LIN {X 0,Y 187.557,Z 471.713,A -85,B 0,C 180,E1 -25907.007,E2 -25907.007} C_VEL
LIN {X 0,Y 185.924,Z 468.386,A -85,B 0,C 180,E1 -25910.069,E2 -25910.069} C_VEL
LIN {X 0,Y 184.642,Z 465.726,A -85,B 0,C 180,E1 -25913.443,E2 -25913.443} C_VEL
LIN {X 0,Y 183.705,Z 463.049,A -85,B 0,C 180,E1 -25920,E2 -25920} C_VEL
LIN {X 0,Y 183.89,Z 463.764,A -85,B 0,C 180,E1 -25923.286,E2 -25923.286} C_VEL
LIN {X 0,Y 185.707,Z 466.949,A -85,B 0,C 180,E1 -25929.53,E2 -25929.53} C_VEL
LIN {X 0,Y 188.183,Z 471.444,A -85,B 0,C 180,E1 -25934.049,E2 -25934.049} C_VEL
LIN {X 0,Y 190.171,Z 475.16,A -85,B 0,C 180,E1 -25936.781,E2 -25936.781} C_VEL
LIN {X 0,Y 192.965,Z 480.658,A -85,B 0,C 180,E1 -25939.965,E2 -25939.965} C_VEL
LIN {X 0,Y 196.223,Z 487.186,A -85,B 0,C 180,E1 -25943.064,E2 -25943.064} C_VEL
LIN {X 0,Y 198.76,Z 492.903,A -85,B 0,C 180,E1 -25945.217,E2 -25945.217} C_VEL
LIN {X 0,Y 191.942,Z 564.548,A -85,B 0,C 180,E1 -25947.122,E2 -25947.122} C_VEL
LIN {X 0,Y 189.485,Z 579.009,A -85,B 0,C 180,E1 -25947.685,E2 -25947.685} C_VEL
LIN {X 0,Y 185.923,Z 593.535,A -85,B 0,C 180,E1 -25948.495,E2 -25948.495} C_VEL
LIN {X 0,Y 181.708,Z 606.777,A -85,B 0,C 180,E1 -25949.514,E2 -25949.514} C_VEL
LIN {X 0,Y 176.215,Z 620.778,A -85,B 0,C 180,E1 -25950.965,E2 -25950.965} C_VEL
LIN {X 0,Y 170.319,Z 633.449,A -85,B 0,C 180,E1 -25952.729,E2 -25952.729} C_VEL
LIN {X 0,Y 163.721,Z 645.382,A -85,B 0,C 180,E1 -25954.818,E2 -25954.818} C_VEL
LIN {X 0,Y 156.791,Z 656.314,A -85,B 0,C 180,E1 -25957.286,E2 -25957.286} C_VEL
LIN {X 0,Y 149.65,Z 666.389,A -85,B 0,C 180,E1 -25960.258,E2 -25960.258} C_VEL
LIN {X 0,Y 141.683,Z 676.375,A -85,B 0,C 180,E1 -25964.143,E2 -25964.143} C_VEL
LIN {X 0,Y 140.976,Z 677.274,A -85,B 0,C 180,E1 -25964.6,E2 -25964.6} C_VEL
LIN {X 0,Y 138.983,Z 679.517,A -85,B 0,C 180,E1 -25965.653,E2 -25965.653} C_VEL
LIN {X 0,Y 135.25,Z 682.744,A -85,B 0,C 180,E1 -25967.021,E2 -25967.021} C_VEL
LIN {X 0,Y 124.177,Z 690.486,A -85,B 0,C 180,E1 -25970.727,E2 -25970.727} C_VEL
LIN {X 0,Y 120.947,Z 693.059,A -85,B 0,C 180,E1 -25972.711,E2 -25972.711} C_VEL
LIN {X 0,Y 114.755,Z 698.936,A -85,B 0,C 180,E1 -25979.026,E2 -25979.026} C_VEL
LIN {X 0,Y 111.351,Z 702.166,A -85,B 0,C 180,E1 -25983.781,E2 -25983.781} C_VEL
LIN {X 0,Y 107.709,Z 705.681,A -85,B 0,C 180,E1 -25990.959,E2 -25990.959} C_VEL
LIN {X 0,Y 105.674,Z 707.991,A -85,B 0,C 180,E1 -25998.492,E2 -25998.492} C_VEL
LIN {X 0,Y 105.023,Z 709.148,A -85,B 0,C 180,E1 -26006.163,E2 -26006.163} C_VEL
LIN {X 0,Y 105.037,Z 709.297,A -85,B 0,C 180,E1 -26010.001,E2 -26010.001} C_VEL
LIN {X 0,Y 105.023,Z 709.143,A -85,B 0,C 180,E1 -26013.838,E2 -26013.838} C_VEL
LIN {X 0,Y 105.675,Z 707.967,A -85,B 0,C 180,E1 -26021.509,E2 -26021.509} C_VEL
LIN {X 0,Y 107.712,Z 705.634,A -85,B 0,C 180,E1 -26029.041,E2 -26029.041} C_VEL
LIN {X 0,Y 111.352,Z 702.088,A -85,B 0,C 180,E1 -26036.22,E2 -26036.22} C_VEL
LIN {X 0,Y 116.463,Z 697.248,A -85,B 0,C 180,E1 -26042.896,E2 -26042.896} C_VEL
LIN {X 0,Y 123.137,Z 690.987,A -85,B 0,C 180,E1 -26048.89,E2 -26048.89} C_VEL
LIN {X 0,Y 130.236,Z 684.232,A -85,B 0,C 180,E1 -26053.475,E2 -26053.475} C_VEL
LIN {X 0,Y 131.674,Z 683.274,A -85,B 0,C 180,E1 -26054.203,E2 -26054.203} C_VEL
LIN {X 0,Y 137.067,Z 683.812,A -85,B 0,C 180,E1 -26056.959,E2 -26056.959} C_VEL
LIN {X 0,Y 137.658,Z 683.754,A -85,B 0,C 180,E1 -26057.806,E2 -26057.806} C_VEL
LIN {X 0,Y 128.187,Z 680.8,A -85,B 0,C 180,E1 -26062.909,E2 -26062.909} C_VEL
LIN {X 0,Y 117.241,Z 675.145,A -85,B 0,C 180,E1 -26071.832,E2 -26071.832} C_VEL
LIN {X 0,Y 112.757,Z 674.144,A -85,B 0,C 180,E1 -26078.04,E2 -26078.04} C_VEL
LIN {X 0,Y 111.56,Z 673.151,A -85,B 0,C 180,E1 -26081.64,E2 -26081.64} C_VEL
LIN {X 0,Y 109.678,Z 671.783,A -85,B 0,C 180,E1 -26088.917,E2 -26088.917} C_VEL
LIN {X 0,Y 110.012,Z 670.647,A -85,B 0,C 180,E1 -26092.66,E2 -26092.66} C_VEL
LIN {X 0,Y 121.004,Z 665.01,A -85,B 0,C 180,E1 -26116.883,E2 -26116.883} C_VEL
LIN {X 0,Y 127.947,Z 662.916,A -85,B 0,C 180,E1 -26122.613,E2 -26122.613} C_VEL
LIN {X 0,Y 140.954,Z 659.025,A -85,B 0,C 180,E1 -26129.908,E2 -26129.908} C_VEL
LIN {X 0,Y 153.456,Z 654.615,A -85,B 0,C 180,E1 -26134.475,E2 -26134.475} C_VEL
LIN {X 0,Y 153.949,Z 654.617,A -85,B 0,C 180,E1 -26134.741,E2 -26134.741} C_VEL
LIN {X 0,Y 146.413,Z 664.975,A -85,B 0,C 180,E1 -26137.624,E2 -26137.624} C_VEL
LIN {X 0,Y 138.047,Z 675.23,A -85,B 0,C 180,E1 -26141.44,E2 -26141.44} C_VEL
LIN {X 0,Y 130.759,Z 683.495,A -85,B 0,C 180,E1 -26145.675,E2 -26145.675} C_VEL
LIN {X 0,Y 124.795,Z 689.57,A -85,B 0,C 180,E1 -26149.635,E2 -26149.635} C_VEL
LIN {X 0,Y 117.999,Z 696.212,A -85,B 0,C 180,E1 -26155.54,E2 -26155.54} C_VEL
LIN {X 0,Y 112.574,Z 701.409,A -85,B 0,C 180,E1 -26162.08,E2 -26162.08} C_VEL
LIN {X 0,Y 109.405,Z 704.399,A -85,B 0,C 180,E1 -26167.329,E2 -26167.329} C_VEL
LIN {X 0,Y 106.519,Z 707.337,A -85,B 0,C 180,E1 -26174.697,E2 -26174.697} C_VEL
LIN {X 0,Y 105.179,Z 709.095,A -85,B 0,C 180,E1 -26182.32,E2 -26182.32} C_VEL
LIN {X 0,Y 105.034,Z 709.702,A -85,B 0,C 180,E1 -26189.999,E2 -26189.999} C_VEL
LIN {X 0,Y 105.17,Z 709.121,A -85,B 0,C 180,E1 -26197.68,E2 -26197.68} C_VEL
LIN {X 0,Y 106.512,Z 707.397,A -85,B 0,C 180,E1 -26205.303,E2 -26205.303} C_VEL
LIN {X 0,Y 109.375,Z 704.501,A -85,B 0,C 180,E1 -26212.677,E2 -26212.677} C_VEL
LIN {X 0,Y 113.686,Z 700.361,A -85,B 0,C 180,E1 -26219.64,E2 -26219.64} C_VEL
LIN {X 0,Y 119.521,Z 694.867,A -85,B 0,C 180,E1 -26226.016,E2 -26226.016} C_VEL
LIN {X 0,Y 126.588,Z 687.87,A -85,B 0,C 180,E1 -26231.776,E2 -26231.776} C_VEL
LIN {X 0,Y 133.805,Z 680.377,A -85,B 0,C 180,E1 -26236.236,E2 -26236.236} C_VEL
LIN {X 0,Y 140.37,Z 672.723,A -85,B 0,C 180,E1 -26239.776,E2 -26239.776} C_VEL
LIN {X 0,Y 147.577,Z 663.733,A -85,B 0,C 180,E1 -26242.909,E2 -26242.909} C_VEL
LIN {X 0,Y 155.109,Z 653.132,A -85,B 0,C 180,E1 -26245.782,E2 -26245.782} C_VEL
LIN {X 0,Y 162.434,Z 641.573,A -85,B 0,C 180,E1 -26248.115,E2 -26248.115} C_VEL
LIN {X 0,Y 169.184,Z 628.933,A -85,B 0,C 180,E1 -26250.14,E2 -26250.14} C_VEL
LIN {X 0,Y 175.433,Z 615.076,A -85,B 0,C 180,E1 -26251.804,E2 -26251.804} C_VEL
LIN {X 0,Y 180.776,Z 600.557,A -85,B 0,C 180,E1 -26253.092,E2 -26253.092} C_VEL
LIN {X 0,Y 185.145,Z 585.35,A -85,B 0,C 180,E1 -26254.048,E2 -26254.048} C_VEL
LIN {X 0,Y 188.341,Z 569.61,A -85,B 0,C 180,E1 -26254.743,E2 -26254.743} C_VEL
LIN {X 0,Y 190.53,Z 551.213,A -85,B 0,C 180,E1 -26255.288,E2 -26255.288} C_VEL
LIN {X 0,Y 195.388,Z 500.881,A -85,B 0,C 180,E1 -26256.558,E2 -26256.558} C_VEL
LIN {X 0,Y 192.605,Z 493.12,A -85,B 0,C 180,E1 -26259.316,E2 -26259.316} C_VEL
LIN {X 0,Y 189.751,Z 486.108,A -85,B 0,C 180,E1 -26262.556,E2 -26262.556} C_VEL
LIN {X 0,Y 187.846,Z 481.849,A -85,B 0,C 180,E1 -26265.095,E2 -26265.095} C_VEL
LIN {X 0,Y 186.025,Z 477.931,A -85,B 0,C 180,E1 -26268.033,E2 -26268.033} C_VEL
LIN {X 0,Y 184.797,Z 475.213,A -85,B 0,C 180,E1 -26270.56,E2 -26270.56} C_VEL
LIN {X 0,Y 183.646,Z 472.659,A -85,B 0,C 180,E1 -26273.821,E2 -26273.821} C_VEL
LIN {X 0,Y 182.834,Z 470.138,A -85,B 0,C 180,E1 -26280,E2 -26280} C_VEL
LIN {X 0,Y 182.964,Z 470.667,A -85,B 0,C 180,E1 -26282.806,E2 -26282.806} C_VEL
LIN {X 0,Y 184.371,Z 473.499,A -85,B 0,C 180,E1 -26288.494,E2 -26288.494} C_VEL
LIN {X 0,Y 185.251,Z 475.089,A -85,B 0,C 180,E1 -26290.52,E2 -26290.52} C_VEL
LIN {X 0,Y 187.03,Z 478.5,A -85,B 0,C 180,E1 -26293.721,E2 -26293.721} C_VEL
LIN {X 0,Y 189.327,Z 483.029,A -85,B 0,C 180,E1 -26296.946,E2 -26296.946} C_VEL
LIN {X 0,Y 192.711,Z 490.116,A -85,B 0,C 180,E1 -26300.758,E2 -26300.758} C_VEL
LIN {X 0,Y 195.47,Z 496.399,A -85,B 0,C 180,E1 -26303.39,E2 -26303.39} C_VEL
LIN {X 0,Y 189.416,Z 559.8,A -85,B 0,C 180,E1 -26305.06,E2 -26305.06} C_VEL
LIN {X 0,Y 187.005,Z 575.537,A -85,B 0,C 180,E1 -26305.583,E2 -26305.583} C_VEL
LIN {X 0,Y 183.72,Z 589.779,A -85,B 0,C 180,E1 -26306.289,E2 -26306.289} C_VEL
LIN {X 0,Y 179.031,Z 604.867,A -85,B 0,C 180,E1 -26307.357,E2 -26307.357} C_VEL
LIN {X 0,Y 174.055,Z 617.673,A -85,B 0,C 180,E1 -26308.572,E2 -26308.572} C_VEL
LIN {X 0,Y 167.915,Z 630.947,A -85,B 0,C 180,E1 -26310.283,E2 -26310.283} C_VEL
LIN {X 0,Y 161.124,Z 643.241,A -85,B 0,C 180,E1 -26312.317,E2 -26312.317} C_VEL
LIN {X 0,Y 153.87,Z 654.478,A -85,B 0,C 180,E1 -26314.7,E2 -26314.7} C_VEL
LIN {X 0,Y 146.369,Z 664.809,A -85,B 0,C 180,E1 -26317.604,E2 -26317.604} C_VEL
LIN {X 0,Y 139.216,Z 673.563,A -85,B 0,C 180,E1 -26320.779,E2 -26320.779} C_VEL
LIN {X 0,Y 132.788,Z 681.059,A -85,B 0,C 180,E1 -26324.398,E2 -26324.398} C_VEL
LIN {X 0,Y 124.748,Z 689.319,A -85,B 0,C 180,E1 -26329.619,E2 -26329.619} C_VEL
LIN {X 0,Y 120.947,Z 693.059,A -85,B 0,C 180,E1 -26332.711,E2 -26332.711} C_VEL
LIN {X 0,Y 117.868,Z 695.504,A -85,B 0,C 180,E1 -26334.852,E2 -26334.852} C_VEL
LIN {X 0,Y 109.03,Z 700.362,A -85,B 0,C 180,E1 -26339.691,E2 -26339.691} C_VEL
LIN {X 0,Y 104.69,Z 702.688,A -85,B 0,C 180,E1 -26343.013,E2 -26343.013} C_VEL
LIN {X 0,Y 103.243,Z 703.671,A -85,B 0,C 180,E1 -26344.944,E2 -26344.944} C_VEL
LIN {X 0,Y 99.65,Z 706.997,A -85,B 0,C 180,E1 -26353.614,E2 -26353.614} C_VEL
LIN {X 0,Y 98.121,Z 708.726,A -85,B 0,C 180,E1 -26361.764,E2 -26361.764} C_VEL
LIN {X 0,Y 97.93,Z 709.161,A -85,B 0,C 180,E1 -26365.885,E2 -26365.885} C_VEL
LIN {X 0,Y 97.944,Z 709.311,A -85,B 0,C 180,E1 -26370.001,E2 -26370.001} C_VEL
LIN {X 0,Y 97.93,Z 709.156,A -85,B 0,C 180,E1 -26374.116,E2 -26374.116} C_VEL
LIN {X 0,Y 98.697,Z 707.98,A -85,B 0,C 180,E1 -26382.335,E2 -26382.335} C_VEL
LIN {X 0,Y 100.976,Z 705.647,A -85,B 0,C 180,E1 -26390.366,E2 -26390.366} C_VEL
LIN {X 0,Y 104.977,Z 702.102,A -85,B 0,C 180,E1 -26397.946,E2 -26397.946} C_VEL
LIN {X 0,Y 110.518,Z 697.262,A -85,B 0,C 180,E1 -26404.913,E2 -26404.913} C_VEL
LIN {X 0,Y 117.662,Z 691.001,A -85,B 0,C 180,E1 -26411.075,E2 -26411.075} C_VEL
LIN {X 0,Y 125.173,Z 684.243,A -85,B 0,C 180,E1 -26415.715,E2 -26415.715} C_VEL
LIN {X 0,Y 127.95,Z 682.049,A -85,B 0,C 180,E1 -26417.039,E2 -26417.039} C_VEL
LIN {X 0,Y 128.251,Z 682.051,A -85,B 0,C 180,E1 -26417.192,E2 -26417.192} C_VEL
LIN {X 0,Y 127.987,Z 681.841,A -85,B 0,C 180,E1 -26417.919,E2 -26417.919} C_VEL
LIN {X 0,Y 123.687,Z 680.797,A -85,B 0,C 180,E1 -26420.266,E2 -26420.266} C_VEL
LIN {X 0,Y 118.591,Z 680.493,A -85,B 0,C 180,E1 -26423.657,E2 -26423.657} C_VEL
LIN {X 0,Y 112.444,Z 679.282,A -85,B 0,C 180,E1 -26429.999,E2 -26429.999} C_VEL
LIN {X 0,Y 107.401,Z 678.331,A -85,B 0,C 180,E1 -26436.883,E2 -26436.883} C_VEL
LIN {X 0,Y 104.1,Z 676.164,A -85,B 0,C 180,E1 -26448.315,E2 -26448.315} C_VEL
LIN {X 0,Y 104.641,Z 674.305,A -85,B 0,C 180,E1 -26456.149,E2 -26456.149} C_VEL
LIN {X 0,Y 119.117,Z 668.837,A -85,B 0,C 180,E1 -26480.733,E2 -26480.733} C_VEL
LIN {X 0,Y 131.561,Z 665.47,A -85,B 0,C 180,E1 -26488.737,E2 -26488.737} C_VEL
LIN {X 0,Y 141.576,Z 662.528,A -85,B 0,C 180,E1 -26493.097,E2 -26493.097} C_VEL
LIN {X 0,Y 144.111,Z 661.736,A -85,B 0,C 180,E1 -26493.997,E2 -26493.997} C_VEL
LIN {X 0,Y 144.749,Z 661.738,A -85,B 0,C 180,E1 -26494.37,E2 -26494.37} C_VEL
LIN {X 0,Y 135.949,Z 672.398,A -85,B 0,C 180,E1 -26497.967,E2 -26497.967} C_VEL
LIN {X 0,Y 129.046,Z 680.084,A -85,B 0,C 180,E1 -26501.509,E2 -26501.509} C_VEL
LIN {X 0,Y 121.42,Z 687.63,A -85,B 0,C 180,E1 -26506.005,E2 -26506.005} C_VEL
LIN {X 0,Y 113.871,Z 694.667,A -85,B 0,C 180,E1 -26511.888,E2 -26511.888} C_VEL
LIN {X 0,Y 107.647,Z 700.2,A -85,B 0,C 180,E1 -26518.513,E2 -26518.513} C_VEL
LIN {X 0,Y 102.839,Z 704.385,A -85,B 0,C 180,E1 -26525.792,E2 -26525.792} C_VEL
LIN {X 0,Y 99.651,Z 707.323,A -85,B 0,C 180,E1 -26533.614,E2 -26533.614} C_VEL
LIN {X 0,Y 98.12,Z 709.082,A -85,B 0,C 180,E1 -26541.763,E2 -26541.763} C_VEL
LIN {X 0,Y 97.941,Z 709.688,A -85,B 0,C 180,E1 -26549.999,E2 -26549.999} C_VEL
LIN {X 0,Y 98.113,Z 709.107,A -85,B 0,C 180,E1 -26558.236,E2 -26558.236} C_VEL
LIN {X 0,Y 99.643,Z 707.383,A -85,B 0,C 180,E1 -26566.387,E2 -26566.387} C_VEL
LIN {X 0,Y 102.807,Z 704.486,A -85,B 0,C 180,E1 -26574.215,E2 -26574.215} C_VEL
LIN {X 0,Y 107.497,Z 700.345,A -85,B 0,C 180,E1 -26581.535,E2 -26581.535} C_VEL
LIN {X 0,Y 113.815,Z 694.85,A -85,B 0,C 180,E1 -26588.133,E2 -26588.133} C_VEL
LIN {X 0,Y 121.352,Z 687.852,A -85,B 0,C 180,E1 -26594.024,E2 -26594.024} C_VEL
LIN {X 0,Y 128.937,Z 680.358,A -85,B 0,C 180,E1 -26598.544,E2 -26598.544} C_VEL
LIN {X 0,Y 137.073,Z 671.326,A -85,B 0,C 180,E1 -26602.628,E2 -26602.628} C_VEL
LIN {X 0,Y 144.681,Z 662.102,A -85,B 0,C 180,E1 -26605.668,E2 -26605.668} C_VEL
LIN {X 0,Y 153.266,Z 650.21,A -85,B 0,C 180,E1 -26608.654,E2 -26608.654} C_VEL
LIN {X 0,Y 160.848,Z 638.067,A -85,B 0,C 180,E1 -26610.911,E2 -26610.911} C_VEL
LIN {X 0,Y 167.877,Z 624.684,A -85,B 0,C 180,E1 -26612.823,E2 -26612.823} C_VEL
LIN {X 0,Y 173.633,Z 611.575,A -85,B 0,C 180,E1 -26614.236,E2 -26614.236} C_VEL
LIN {X 0,Y 178.792,Z 597.21,A -85,B 0,C 180,E1 -26615.367,E2 -26615.367} C_VEL
LIN {X 0,Y 182.898,Z 582.338,A -85,B 0,C 180,E1 -26616.207,E2 -26616.207} C_VEL
LIN {X 0,Y 185.886,Z 566.815,A -85,B 0,C 180,E1 -26616.817,E2 -26616.817} C_VEL
LIN {X 0,Y 189.95,Z 528.58,A -85,B 0,C 180,E1 -26617.779,E2 -26617.779} C_VEL
LIN {X 0,Y 192.33,Z 504.169,A -85,B 0,C 180,E1 -26618.412,E2 -26618.412} C_VEL
LIN {X 0,Y 189.556,Z 496.227,A -85,B 0,C 180,E1 -26621.527,E2 -26621.527} C_VEL
LIN {X 0,Y 186.843,Z 489.339,A -85,B 0,C 180,E1 -26625.152,E2 -26625.152} C_VEL
LIN {X 0,Y 184.873,Z 484.832,A -85,B 0,C 180,E1 -26628.451,E2 -26628.451} C_VEL
LIN {X 0,Y 183.522,Z 481.695,A -85,B 0,C 180,E1 -26631.466,E2 -26631.466} C_VEL
LIN {X 0,Y 182.585,Z 479.467,A -85,B 0,C 180,E1 -26634.478,E2 -26634.478} C_VEL
LIN {X 0,Y 181.964,Z 477.224,A -85,B 0,C 180,E1 -26640,E2 -26640} C_VEL
LIN {X 0,Y 182.09,Z 477.732,A -85,B 0,C 180,E1 -26642.765,E2 -26642.765} C_VEL
LIN {X 0,Y 183.706,Z 480.982,A -85,B 0,C 180,E1 -26649.036,E2 -26649.036} C_VEL
LIN {X 0,Y 185.598,Z 484.944,A -85,B 0,C 180,E1 -26652.907,E2 -26652.907} C_VEL
LIN {X 0,Y 187.679,Z 489.286,A -85,B 0,C 180,E1 -26656.068,E2 -26656.068} C_VEL
LIN {X 0,Y 190.791,Z 496.28,A -85,B 0,C 180,E1 -26659.851,E2 -26659.851} C_VEL
LIN {X 0,Y 192.425,Z 500.192,A -85,B 0,C 180,E1 -26661.562,E2 -26661.562} C_VEL
LIN {X 0,Y 186.194,Z 562.512,A -85,B 0,C 180,E1 -26663.163,E2 -26663.163} C_VEL
LIN {X 0,Y 183.686,Z 577.382,A -85,B 0,C 180,E1 -26663.671,E2 -26663.671} C_VEL
LIN {X 0,Y 179.963,Z 592.37,A -85,B 0,C 180,E1 -26664.438,E2 -26664.438} C_VEL
LIN {X 0,Y 175.151,Z 606.859,A -85,B 0,C 180,E1 -26665.469,E2 -26665.469} C_VEL
LIN {X 0,Y 169.339,Z 620.846,A -85,B 0,C 180,E1 -26666.836,E2 -26666.836} C_VEL
LIN {X 0,Y 162.674,Z 634.228,A -85,B 0,C 180,E1 -26668.633,E2 -26668.633} C_VEL
LIN {X 0,Y 155.346,Z 646.49,A -85,B 0,C 180,E1 -26670.732,E2 -26670.732} C_VEL
LIN {X 0,Y 147.265,Z 658.124,A -85,B 0,C 180,E1 -26673.368,E2 -26673.368} C_VEL
LIN {X 0,Y 139.601,Z 667.908,A -85,B 0,C 180,E1 -26676.342,E2 -26676.342} C_VEL
LIN {X 0,Y 131.111,Z 677.472,A -85,B 0,C 180,E1 -26680.196,E2 -26680.196} C_VEL
LIN {X 0,Y 124.595,Z 684.398,A -85,B 0,C 180,E1 -26684.013,E2 -26684.013} C_VEL
LIN {X 0,Y 117.454,Z 691.133,A -85,B 0,C 180,E1 -26688.838,E2 -26688.838} C_VEL
LIN {X 0,Y 110.492,Z 697.371,A -85,B 0,C 180,E1 -26695.079,E2 -26695.079} C_VEL
LIN {X 0,Y 104.978,Z 702.182,A -85,B 0,C 180,E1 -26702.055,E2 -26702.055} C_VEL
LIN {X 0,Y 103.243,Z 703.671,A -85,B 0,C 180,E1 -26704.944,E2 -26704.944} C_VEL
LIN {X 0,Y 101.084,Z 705.115,A -85,B 0,C 180,E1 -26707.918,E2 -26707.918} C_VEL
LIN {X 0,Y 96.328,Z 707.026,A -85,B 0,C 180,E1 -26712.844,E2 -26712.844} C_VEL
LIN {X 0,Y 92.819,Z 708.119,A -85,B 0,C 180,E1 -26717.134,E2 -26717.134} C_VEL
LIN {X 0,Y 91.217,Z 708.691,A -85,B 0,C 180,E1 -26720.681,E2 -26720.681} C_VEL
LIN {X 0,Y 91,Z 708.818,A -85,B 0,C 180,E1 -26721.916,E2 -26721.916} C_VEL
LIN {X 0,Y 90.843,Z 709.324,A -85,B 0,C 180,E1 -26730.001,E2 -26730.001} C_VEL
LIN {X 0,Y 90.83,Z 709.17,A -85,B 0,C 180,E1 -26734.438,E2 -26734.438} C_VEL
LIN {X 0,Y 91.753,Z 707.994,A -85,B 0,C 180,E1 -26743.285,E2 -26743.285} C_VEL
LIN {X 0,Y 94.301,Z 705.661,A -85,B 0,C 180,E1 -26751.879,E2 -26751.879} C_VEL
LIN {X 0,Y 98.716,Z 702.115,A -85,B 0,C 180,E1 -26759.892,E2 -26759.892} C_VEL
LIN {X 0,Y 104.732,Z 697.276,A -85,B 0,C 180,E1 -26767.153,E2 -26767.153} C_VEL
LIN {X 0,Y 112.382,Z 691.015,A -85,B 0,C 180,E1 -26773.465,E2 -26773.465} C_VEL
LIN {X 0,Y 119.107,Z 685.31,A -85,B 0,C 180,E1 -26777.507,E2 -26777.507} C_VEL
LIN {X 0,Y 118.001,Z 684.542,A -85,B 0,C 180,E1 -26779.07,E2 -26779.07} C_VEL
LIN {X 0,Y 113.824,Z 684.316,A -85,B 0,C 180,E1 -26781.871,E2 -26781.871} C_VEL
LIN {X 0,Y 104.328,Z 682.804,A -85,B 0,C 180,E1 -26791.865,E2 -26791.865} C_VEL
LIN {X 0,Y 101.937,Z 682.31,A -85,B 0,C 180,E1 -26795.565,E2 -26795.565} C_VEL
LIN {X 0,Y 98.331,Z 680.275,A -85,B 0,C 180,E1 -26807.619,E2 -26807.619} C_VEL
LIN {X 0,Y 99.648,Z 677.815,A -85,B 0,C 180,E1 -26820,E2 -26820} C_VEL
LIN {X 0,Y 113.887,Z 673.365,A -85,B 0,C 180,E1 -26841.732,E2 -26841.732} C_VEL
LIN {X 0,Y 126.706,Z 670.234,A -85,B 0,C 180,E1 -26849.948,E2 -26849.948} C_VEL
LIN {X 0,Y 135.535,Z 668.037,A -85,B 0,C 180,E1 -26853.935,E2 -26853.935} C_VEL
LIN {X 0,Y 126.952,Z 677.401,A -85,B 0,C 180,E1 -26857.677,E2 -26857.677} C_VEL
LIN {X 0,Y 119.812,Z 684.572,A -85,B 0,C 180,E1 -26861.591,E2 -26861.591} C_VEL
LIN {X 0,Y 112.207,Z 691.335,A -85,B 0,C 180,E1 -26866.45,E2 -26866.45} C_VEL
LIN {X 0,Y 104.784,Z 697.596,A -85,B 0,C 180,E1 -26872.868,E2 -26872.868} C_VEL
LIN {X 0,Y 98.776,Z 702.44,A -85,B 0,C 180,E1 -26880.128,E2 -26880.128} C_VEL
LIN {X 0,Y 94.322,Z 705.992,A -85,B 0,C 180,E1 -26888.126,E2 -26888.126} C_VEL
LIN {X 0,Y 91.753,Z 708.333,A -85,B 0,C 180,E1 -26896.715,E2 -26896.715} C_VEL
LIN {X 0,Y 90.8,Z 709.518,A -85,B 0,C 180,E1 -26905.56,E2 -26905.56} C_VEL
LIN {X 0,Y 90.841,Z 709.675,A -85,B 0,C 180,E1 -26909.999,E2 -26909.999} C_VEL
LIN {X 0,Y 91.08,Z 709.093,A -85,B 0,C 180,E1 -26918.877,E2 -26918.877} C_VEL
LIN {X 0,Y 92.822,Z 707.369,A -85,B 0,C 180,E1 -26927.629,E2 -26927.629} C_VEL
LIN {X 0,Y 96.328,Z 704.471,A -85,B 0,C 180,E1 -26935.96,E2 -26935.96} C_VEL
LIN {X 0,Y 101.646,Z 700.148,A -85,B 0,C 180,E1 -26943.931,E2 -26943.931} C_VEL
LIN {X 0,Y 108.26,Z 694.834,A -85,B 0,C 180,E1 -26950.479,E2 -26950.479} C_VEL
LIN {X 0,Y 116.328,Z 687.835,A -85,B 0,C 180,E1 -26956.467,E2 -26956.467} C_VEL
LIN {X 0,Y 123.166,Z 681.497,A -85,B 0,C 180,E1 -26960.383,E2 -26960.383} C_VEL
LIN {X 0,Y 131.582,Z 672.683,A -85,B 0,C 180,E1 -26964.54,E2 -26964.54} C_VEL
LIN {X 0,Y 139.43,Z 663.691,A -85,B 0,C 180,E1 -26967.595,E2 -26967.595} C_VEL
LIN {X 0,Y 147.582,Z 653.085,A -85,B 0,C 180,E1 -26970.351,E2 -26970.351} C_VEL
LIN {X 0,Y 155.38,Z 641.519,A -85,B 0,C 180,E1 -26972.58,E2 -26972.58} C_VEL
LIN {X 0,Y 162.281,Z 629.415,A -85,B 0,C 180,E1 -26974.427,E2 -26974.427} C_VEL
LIN {X 0,Y 168.441,Z 616.732,A -85,B 0,C 180,E1 -26975.882,E2 -26975.882} C_VEL
LIN {X 0,Y 174.056,Z 602.665,A -85,B 0,C 180,E1 -26977.09,E2 -26977.09} C_VEL
LIN {X 0,Y 178.63,Z 588.174,A -85,B 0,C 180,E1 -26977.978,E2 -26977.978} C_VEL
LIN {X 0,Y 182.16,Z 572.756,A -85,B 0,C 180,E1 -26978.653,E2 -26978.653} C_VEL
LIN {X 0,Y 184.496,Z 556.413,A -85,B 0,C 180,E1 -26979.142,E2 -26979.142} C_VEL
LIN {X 0,Y 189.448,Z 507.557,A -85,B 0,C 180,E1 -26980.341,E2 -26980.341} C_VEL
LIN {X 0,Y 187.399,Z 501.513,A -85,B 0,C 180,E1 -26982.912,E2 -26982.912} C_VEL
LIN {X 0,Y 185.313,Z 495.698,A -85,B 0,C 180,E1 -26986.009,E2 -26986.009} C_VEL
LIN {X 0,Y 183.422,Z 491.038,A -85,B 0,C 180,E1 -26989.513,E2 -26989.513} C_VEL
LIN {X 0,Y 182.255,Z 488.018,A -85,B 0,C 180,E1 -26992.522,E2 -26992.522} C_VEL
LIN {X 0,Y 181.521,Z 486.185,A -85,B 0,C 180,E1 -26995.28,E2 -26995.28} C_VEL
LIN {X 0,Y 181.094,Z 484.311,A -85,B 0,C 180,E1 -27000,E2 -27000} C_VEL
LIN {X 0,Y 181.221,Z 484.813,A -85,B 0,C 180,E1 -27002.778,E2 -27002.778} C_VEL
LIN {X 0,Y 182.679,Z 487.972,A -85,B 0,C 180,E1 -27008.713,E2 -27008.713} C_VEL
LIN {X 0,Y 184.456,Z 491.931,A -85,B 0,C 180,E1 -27012.542,E2 -27012.542} C_VEL
LIN {X 0,Y 186.616,Z 496.91,A -85,B 0,C 180,E1 -27015.97,E2 -27015.97} C_VEL
LIN {X 0,Y 189.572,Z 503.969,A -85,B 0,C 180,E1 -27019.667,E2 -27019.667} C_VEL
LIN {X 0,Y 183.191,Z 565.066,A -85,B 0,C 180,E1 -27021.187,E2 -27021.187} C_VEL
LIN {X 0,Y 180.597,Z 579.224,A -85,B 0,C 180,E1 -27021.705,E2 -27021.705} C_VEL
LIN {X 0,Y 176.767,Z 593.692,A -85,B 0,C 180,E1 -27022.425,E2 -27022.425} C_VEL
LIN {X 0,Y 172.217,Z 606.901,A -85,B 0,C 180,E1 -27023.336,E2 -27023.336} C_VEL
LIN {X 0,Y 166.246,Z 620.881,A -85,B 0,C 180,E1 -27024.646,E2 -27024.646} C_VEL
LIN {X 0,Y 159.166,Z 634.654,A -85,B 0,C 180,E1 -27026.448,E2 -27026.448} C_VEL
LIN {X 0,Y 151.84,Z 646.515,A -85,B 0,C 180,E1 -27028.428,E2 -27028.428} C_VEL
LIN {X 0,Y 143.475,Z 658.147,A -85,B 0,C 180,E1 -27030.994,E2 -27030.994} C_VEL
LIN {X 0,Y 135.488,Z 667.929,A -85,B 0,C 180,E1 -27033.907,E2 -27033.907} C_VEL
LIN {X 0,Y 127.097,Z 676.981,A -85,B 0,C 180,E1 -27037.464,E2 -27037.464} C_VEL
LIN {X 0,Y 119.747,Z 684.416,A -85,B 0,C 180,E1 -27041.557,E2 -27041.557} C_VEL
LIN {X 0,Y 112.169,Z 691.15,A -85,B 0,C 180,E1 -27046.433,E2 -27046.433} C_VEL
LIN {X 0,Y 104.705,Z 697.387,A -85,B 0,C 180,E1 -27052.837,E2 -27052.837} C_VEL
LIN {X 0,Y 98.718,Z 702.197,A -85,B 0,C 180,E1 -27060.11,E2 -27060.11} C_VEL
LIN {X 0,Y 94.298,Z 705.711,A -85,B 0,C 180,E1 -27068.121,E2 -27068.121} C_VEL
LIN {X 0,Y 91.753,Z 708.019,A -85,B 0,C 180,E1 -27076.716,E2 -27076.716} C_VEL
LIN {X 0,Y 91,Z 708.818,A -85,B 0,C 180,E1 -27081.916,E2 -27081.916} C_VEL
LIN {X 0,Y 90.041,Z 709.179,A -85,B 0,C 180,E1 -27085.599,E2 -27085.599} C_VEL
LIN {X 0,Y 88.319,Z 709.313,A -85,B 0,C 180,E1 -27089.26,E2 -27089.26} C_VEL
LIN {X 0,Y 84.853,Z 708.996,A -85,B 0,C 180,E1 -27096.908,E2 -27096.908} C_VEL
LIN {X 0,Y 84.278,Z 708.578,A -85,B 0,C 180,E1 -27100.958,E2 -27100.958} C_VEL
LIN {X 0,Y 84.409,Z 708.328,A -85,B 0,C 180,E1 -27102.311,E2 -27102.311} C_VEL
LIN {X 0,Y 86.042,Z 706.988,A -85,B 0,C 180,E1 -27109.071,E2 -27109.071} C_VEL
LIN {X 0,Y 89.952,Z 704.057,A -85,B 0,C 180,E1 -27117.956,E2 -27117.956} C_VEL
LIN {X 0,Y 95.696,Z 699.815,A -85,B 0,C 180,E1 -27126.114,E2 -27126.114} C_VEL
LIN {X 0,Y 103.036,Z 694.347,A -85,B 0,C 180,E1 -27133.008,E2 -27133.008} C_VEL
LIN {X 0,Y 109.3,Z 689.476,A -85,B 0,C 180,E1 -27137.318,E2 -27137.318} C_VEL
LIN {X 0,Y 110.212,Z 687.914,A -85,B 0,C 180,E1 -27139.081,E2 -27139.081} C_VEL
LIN {X 0,Y 104.363,Z 687.333,A -85,B 0,C 180,E1 -27143.912,E2 -27143.912} C_VEL
LIN {X 0,Y 96.419,Z 686.021,A -85,B 0,C 180,E1 -27154.066,E2 -27154.066} C_VEL
LIN {X 0,Y 92.341,Z 683.338,A -85,B 0,C 180,E1 -27171.245,E2 -27171.245} C_VEL
LIN {X 0,Y 96.796,Z 680.537,A -85,B 0,C 180,E1 -27188.35,E2 -27188.35} C_VEL
LIN {X 0,Y 108.523,Z 677.662,A -85,B 0,C 180,E1 -27202.866,E2 -27202.866} C_VEL
LIN {X 0,Y 124.258,Z 674.179,A -85,B 0,C 180,E1 -27212.502,E2 -27212.502} C_VEL
LIN {X 0,Y 125.526,Z 673.895,A -85,B 0,C 180,E1 -27213.086,E2 -27213.086} C_VEL
LIN {X 0,Y 124.864,Z 675.223,A -85,B 0,C 180,E1 -27214.067,E2 -27214.067} C_VEL
LIN {X 0,Y 116.397,Z 683.452,A -85,B 0,C 180,E1 -27218.285,E2 -27218.285} C_VEL
LIN {X 0,Y 109.308,Z 689.527,A -85,B 0,C 180,E1 -27222.319,E2 -27222.319} C_VEL
LIN {X 0,Y 101.037,Z 696.17,A -85,B 0,C 180,E1 -27228.638,E2 -27228.638} C_VEL
LIN {X 0,Y 94.147,Z 701.368,A -85,B 0,C 180,E1 -27235.953,E2 -27235.953} C_VEL
LIN {X 0,Y 89.992,Z 704.358,A -85,B 0,C 180,E1 -27242.057,E2 -27242.057} C_VEL
LIN {X 0,Y 86.047,Z 707.296,A -85,B 0,C 180,E1 -27250.93,E2 -27250.93} C_VEL
LIN {X 0,Y 84.052,Z 709.054,A -85,B 0,C 180,E1 -27260.373,E2 -27260.373} C_VEL
LIN {X 0,Y 83.762,Z 709.661,A -85,B 0,C 180,E1 -27269.999,E2 -27269.999} C_VEL
LIN {X 0,Y 84.047,Z 709.079,A -85,B 0,C 180,E1 -27279.627,E2 -27279.627} C_VEL
LIN {X 0,Y 86.037,Z 707.354,A -85,B 0,C 180,E1 -27289.071,E2 -27289.071} C_VEL
LIN {X 0,Y 89.957,Z 704.456,A -85,B 0,C 180,E1 -27297.953,E2 -27297.953} C_VEL
LIN {X 0,Y 95.559,Z 700.314,A -85,B 0,C 180,E1 -27306.041,E2 -27306.041} C_VEL
LIN {X 0,Y 102.921,Z 694.817,A -85,B 0,C 180,E1 -27313.067,E2 -27313.067} C_VEL
LIN {X 0,Y 111.539,Z 687.817,A -85,B 0,C 180,E1 -27319.122,E2 -27319.122} C_VEL
LIN {X 0,Y 118.71,Z 681.479,A -85,B 0,C 180,E1 -27323.057,E2 -27323.057} C_VEL
LIN {X 0,Y 127.572,Z 672.664,A -85,B 0,C 180,E1 -27327.153,E2 -27327.153} C_VEL
LIN {X 0,Y 135.741,Z 663.669,A -85,B 0,C 180,E1 -27330.138,E2 -27330.138} C_VEL
LIN {X 0,Y 144.198,Z 653.061,A -85,B 0,C 180,E1 -27332.807,E2 -27332.807} C_VEL
LIN {X 0,Y 152.223,Z 641.492,A -85,B 0,C 180,E1 -27334.967,E2 -27334.967} C_VEL
LIN {X 0,Y 159.746,Z 628.619,A -85,B 0,C 180,E1 -27336.831,E2 -27336.831} C_VEL
LIN {X 0,Y 166.419,Z 614.965,A -85,B 0,C 180,E1 -27338.29,E2 -27338.29} C_VEL
LIN {X 0,Y 172.19,Z 600.419,A -85,B 0,C 180,E1 -27339.423,E2 -27339.423} C_VEL
LIN {X 0,Y 176.875,Z 585.168,A -85,B 0,C 180,E1 -27340.255,E2 -27340.255} C_VEL
LIN {X 0,Y 180.179,Z 569.988,A -85,B 0,C 180,E1 -27340.847,E2 -27340.847} C_VEL
LIN {X 0,Y 182.411,Z 553.072,A -85,B 0,C 180,E1 -27341.317,E2 -27341.317} C_VEL
LIN {X 0,Y 186.792,Z 511.201,A -85,B 0,C 180,E1 -27342.291,E2 -27342.291} C_VEL
LIN {X 0,Y 185.055,Z 505.853,A -85,B 0,C 180,E1 -27344.794,E2 -27344.794} C_VEL
LIN {X 0,Y 183.539,Z 501.335,A -85,B 0,C 180,E1 -27347.388,E2 -27347.388} C_VEL
LIN {X 0,Y 182.106,Z 497.425,A -85,B 0,C 180,E1 -27350.419,E2 -27350.419} C_VEL
LIN {X 0,Y 181.116,Z 494.636,A -85,B 0,C 180,E1 -27353.315,E2 -27353.315} C_VEL
LIN {X 0,Y 180.515,Z 492.975,A -85,B 0,C 180,E1 -27355.953,E2 -27355.953} C_VEL
LIN {X 0,Y 180.224,Z 491.396,A -85,B 0,C 180,E1 -27360,E2 -27360} C_VEL
LIN {X 0,Y 180.338,Z 491.855,A -85,B 0,C 180,E1 -27362.652,E2 -27362.652} C_VEL
LIN {X 0,Y 181.595,Z 494.816,A -85,B 0,C 180,E1 -27368.205,E2 -27368.205} C_VEL
LIN {X 0,Y 183.143,Z 498.53,A -85,B 0,C 180,E1 -27371.833,E2 -27371.833} C_VEL
LIN {X 0,Y 185.058,Z 503.289,A -85,B 0,C 180,E1 -27375.135,E2 -27375.135} C_VEL
LIN {X 0,Y 186.902,Z 507.979,A -85,B 0,C 180,E1 -27377.714,E2 -27377.714} C_VEL
LIN {X 0,Y 180.829,Z 564.621,A -85,B 0,C 180,E1 -27379.08,E2 -27379.08} C_VEL
LIN {X 0,Y 178.275,Z 578.411,A -85,B 0,C 180,E1 -27379.536,E2 -27379.536} C_VEL
LIN {X 0,Y 174.183,Z 593.743,A -85,B 0,C 180,E1 -27380.265,E2 -27380.265} C_VEL
LIN {X 0,Y 169.537,Z 606.942,A -85,B 0,C 180,E1 -27381.138,E2 -27381.138} C_VEL
LIN {X 0,Y 163.416,Z 620.915,A -85,B 0,C 180,E1 -27382.386,E2 -27382.386} C_VEL
LIN {X 0,Y 156.281,Z 634.407,A -85,B 0,C 180,E1 -27384.064,E2 -27384.064} C_VEL
LIN {X 0,Y 148.589,Z 646.541,A -85,B 0,C 180,E1 -27386.017,E2 -27386.017} C_VEL
LIN {X 0,Y 139.946,Z 658.169,A -85,B 0,C 180,E1 -27388.498,E2 -27388.498} C_VEL
LIN {X 0,Y 131.635,Z 667.95,A -85,B 0,C 180,E1 -27391.325,E2 -27391.325} C_VEL
LIN {X 0,Y 122.374,Z 677.486,A -85,B 0,C 180,E1 -27395.05,E2 -27395.05} C_VEL
LIN {X 0,Y 115.121,Z 684.434,A -85,B 0,C 180,E1 -27398.889,E2 -27398.889} C_VEL
LIN {X 0,Y 107.093,Z 691.167,A -85,B 0,C 180,E1 -27403.791,E2 -27403.791} C_VEL
LIN {X 0,Y 99.087,Z 697.403,A -85,B 0,C 180,E1 -27410.332,E2 -27410.332} C_VEL
LIN {X 0,Y 92.591,Z 702.212,A -85,B 0,C 180,E1 -27417.906,E2 -27417.906} C_VEL
LIN {X 0,Y 87.704,Z 705.725,A -85,B 0,C 180,E1 -27426.381,E2 -27426.381} C_VEL
LIN {X 0,Y 84.817,Z 708.034,A -85,B 0,C 180,E1 -27435.607,E2 -27435.607} C_VEL
LIN {X 0,Y 83.754,Z 709.189,A -85,B 0,C 180,E1 -27445.187,E2 -27445.187} C_VEL
LIN {X 0,Y 83.764,Z 709.338,A -85,B 0,C 180,E1 -27450.001,E2 -27450.001} C_VEL
LIN {X 0,Y 83.754,Z 709.184,A -85,B 0,C 180,E1 -27454.814,E2 -27454.814} C_VEL
LIN {X 0,Y 84.409,Z 708.328,A -85,B 0,C 180,E1 -27462.311,E2 -27462.311} C_VEL
LIN {X 0,Y 84.574,Z 707.687,A -85,B 0,C 180,E1 -27466.283,E2 -27466.283} C_VEL
LIN {X 0,Y 83.815,Z 706.19,A -85,B 0,C 180,E1 -27472.934,E2 -27472.934} C_VEL
LIN {X 0,Y 83.79,Z 704.692,A -85,B 0,C 180,E1 -27478.283,E2 -27478.283} C_VEL
LIN {X 0,Y 85.292,Z 703.068,A -85,B 0,C 180,E1 -27482.722,E2 -27482.722} C_VEL
LIN {X 0,Y 85.673,Z 702.732,A -85,B 0,C 180,E1 -27483.31,E2 -27483.31} C_VEL
LIN {X 0,Y 91.767,Z 698.659,A -85,B 0,C 180,E1 -27490.616,E2 -27490.616} C_VEL
LIN {X 0,Y 100.176,Z 692.762,A -85,B 0,C 180,E1 -27497.447,E2 -27497.447} C_VEL
LIN {X 0,Y 102.513,Z 691.043,A -85,B 0,C 180,E1 -27498.95,E2 -27498.95} C_VEL
LIN {X 0,Y 90.836,Z 689.485,A -85,B 0,C 180,E1 -27512.341,E2 -27512.341} C_VEL
LIN {X 0,Y 86.18,Z 687.036,A -85,B 0,C 180,E1 -27530.614,E2 -27530.614} C_VEL
LIN {X 0,Y 90.774,Z 684.395,A -85,B 0,C 180,E1 -27548.908,E2 -27548.908} C_VEL
LIN {X 0,Y 103.05,Z 681.714,A -85,B 0,C 180,E1 -27564.155,E2 -27564.155} C_VEL
LIN {X 0,Y 116.736,Z 679.012,A -85,B 0,C 180,E1 -27572.809,E2 -27572.809} C_VEL
LIN {X 0,Y 114.629,Z 681.223,A -85,B 0,C 180,E1 -27574.137,E2 -27574.137} C_VEL
LIN {X 0,Y 107.066,Z 687.588,A -85,B 0,C 180,E1 -27578.028,E2 -27578.028} C_VEL
LIN {X 0,Y 97.878,Z 694.625,A -85,B 0,C 180,E1 -27584.106,E2 -27584.106} C_VEL
LIN {X 0,Y 90.035,Z 700.159,A -85,B 0,C 180,E1 -27591.356,E2 -27591.356} C_VEL
LIN {X 0,Y 83.752,Z 704.345,A -85,B 0,C 180,E1 -27599.768,E2 -27599.768} C_VEL
LIN {X 0,Y 79.313,Z 707.283,A -85,B 0,C 180,E1 -27609.24,E2 -27609.24} C_VEL
LIN {X 0,Y 77.046,Z 709.041,A -85,B 0,C 180,E1 -27619.488,E2 -27619.488} C_VEL
LIN {X 0,Y 76.673,Z 709.647,A -85,B 0,C 180,E1 -27629.999,E2 -27629.999} C_VEL
LIN {X 0,Y 77.042,Z 709.065,A -85,B 0,C 180,E1 -27640.512,E2 -27640.512} C_VEL
LIN {X 0,Y 79.302,Z 707.34,A -85,B 0,C 180,E1 -27650.762,E2 -27650.762} C_VEL
LIN {X 0,Y 83.715,Z 704.441,A -85,B 0,C 180,E1 -27660.245,E2 -27660.245} C_VEL
LIN {X 0,Y 89.882,Z 700.298,A -85,B 0,C 180,E1 -27668.72,E2 -27668.72} C_VEL
LIN {X 0,Y 97.804,Z 694.801,A -85,B 0,C 180,E1 -27675.937,E2 -27675.937} C_VEL
LIN {X 0,Y 107.016,Z 687.8,A -85,B 0,C 180,E1 -27682.005,E2 -27682.005} C_VEL
LIN {X 0,Y 115.797,Z 680.301,A -85,B 0,C 180,E1 -27686.565,E2 -27686.565} C_VEL
LIN {X 0,Y 125.224,Z 671.265,A -85,B 0,C 180,E1 -27690.448,E2 -27690.448} C_VEL
LIN {X 0,Y 133.771,Z 662.037,A -85,B 0,C 180,E1 -27693.269,E2 -27693.269} C_VEL
LIN {X 0,Y 143.31,Z 650.136,A -85,B 0,C 180,E1 -27695.976,E2 -27695.976} C_VEL
LIN {X 0,Y 151.616,Z 637.983,A -85,B 0,C 180,E1 -27697.984,E2 -27697.984} C_VEL
LIN {X 0,Y 159.26,Z 624.585,A -85,B 0,C 180,E1 -27699.675,E2 -27699.675} C_VEL
LIN {X 0,Y 165.478,Z 611.46,A -85,B 0,C 180,E1 -27700.904,E2 -27700.904} C_VEL
LIN {X 0,Y 171.008,Z 597.065,A -85,B 0,C 180,E1 -27701.875,E2 -27701.875} C_VEL
LIN {X 0,Y 175.403,Z 582.145,A -85,B 0,C 180,E1 -27702.574,E2 -27702.574} C_VEL
LIN {X 0,Y 178.632,Z 566.121,A -85,B 0,C 180,E1 -27703.121,E2 -27703.121} C_VEL
LIN {X 0,Y 183.446,Z 523.665,A -85,B 0,C 180,E1 -27704.059,E2 -27704.059} C_VEL
LIN {X 0,Y 184.317,Z 514.847,A -85,B 0,C 180,E1 -27704.339,E2 -27704.339} C_VEL
LIN {X 0,Y 182.369,Z 508.362,A -85,B 0,C 180,E1 -27707.789,E2 -27707.789} C_VEL
LIN {X 0,Y 180.885,Z 503.969,A -85,B 0,C 180,E1 -27711.2,E2 -27711.2} C_VEL
LIN {X 0,Y 180.082,Z 501.463,A -85,B 0,C 180,E1 -27713.839,E2 -27713.839} C_VEL
LIN {X 0,Y 179.574,Z 499.905,A -85,B 0,C 180,E1 -27716.353,E2 -27716.353} C_VEL
LIN {X 0,Y 179.354,Z 498.483,A -85,B 0,C 180,E1 -27720,E2 -27720} C_VEL
LIN {X 0,Y 179.433,Z 498.806,A -85,B 0,C 180,E1 -27722.244,E2 -27722.244} C_VEL
LIN {X 0,Y 180.523,Z 501.67,A -85,B 0,C 180,E1 -27727.691,E2 -27727.691} C_VEL
LIN {X 0,Y 181.87,Z 505.162,A -85,B 0,C 180,E1 -27731.14,E2 -27731.14} C_VEL
LIN {X 0,Y 183.574,Z 509.732,A -85,B 0,C 180,E1 -27734.338,E2 -27734.338} C_VEL
LIN {X 0,Y 184.442,Z 512.24,A -85,B 0,C 180,E1 -27735.728,E2 -27735.728} C_VEL
LIN {X 0,Y 178.531,Z 565.511,A -85,B 0,C 180,E1 -27736.951,E2 -27736.951} C_VEL
LIN {X 0,Y 175.841,Z 579.367,A -85,B 0,C 180,E1 -27737.402,E2 -27737.402} C_VEL
LIN {X 0,Y 171.849,Z 593.795,A -85,B 0,C 180,E1 -27738.041,E2 -27738.041} C_VEL
LIN {X 0,Y 167.107,Z 606.982,A -85,B 0,C 180,E1 -27738.866,E2 -27738.866} C_VEL
LIN {X 0,Y 160.841,Z 620.948,A -85,B 0,C 180,E1 -27740.042,E2 -27740.042} C_VEL
LIN {X 0,Y 153.725,Z 634.084,A -85,B 0,C 180,E1 -27741.589,E2 -27741.589} C_VEL
LIN {X 0,Y 145.602,Z 646.566,A -85,B 0,C 180,E1 -27743.495,E2 -27743.495} C_VEL
LIN {X 0,Y 136.695,Z 658.192,A -85,B 0,C 180,E1 -27745.877,E2 -27745.877} C_VEL
LIN {X 0,Y 128.08,Z 667.97,A -85,B 0,C 180,E1 -27748.605,E2 -27748.605} C_VEL
LIN {X 0,Y 119.751,Z 676.309,A -85,B 0,C 180,E1 -27751.685,E2 -27751.685} C_VEL
LIN {X 0,Y 110.778,Z 684.451,A -85,B 0,C 180,E1 -27756.013,E2 -27756.013} C_VEL
LIN {X 0,Y 102.273,Z 691.183,A -85,B 0,C 180,E1 -27760.897,E2 -27760.897} C_VEL
LIN {X 0,Y 93.694,Z 697.419,A -85,B 0,C 180,E1 -27767.539,E2 -27767.539} C_VEL
LIN {X 0,Y 86.617,Z 702.227,A -85,B 0,C 180,E1 -27775.392,E2 -27775.392} C_VEL
LIN {X 0,Y 81.211,Z 705.74,A -85,B 0,C 180,E1 -27784.362,E2 -27784.362} C_VEL
LIN {X 0,Y 77.928,Z 708.048,A -85,B 0,C 180,E1 -27794.303,E2 -27794.303} C_VEL
LIN {X 0,Y 76.657,Z 709.203,A -85,B 0,C 180,E1 -27804.74,E2 -27804.74} C_VEL
LIN {X 0,Y 76.675,Z 709.352,A -85,B 0,C 180,E1 -27810.001,E2 -27810.001} C_VEL
LIN {X 0,Y 77.046,Z 708.751,A -85,B 0,C 180,E1 -27820.512,E2 -27820.512} C_VEL
LIN {X 0,Y 79.307,Z 707.002,A -85,B 0,C 180,E1 -27830.762,E2 -27830.762} C_VEL
LIN {X 0,Y 83.712,Z 704.071,A -85,B 0,C 180,E1 -27840.248,E2 -27840.248} C_VEL
LIN {X 0,Y 85.673,Z 702.732,A -85,B 0,C 180,E1 -27843.31,E2 -27843.31} C_VEL
LIN {X 0,Y 86.73,Z 701.696,A -85,B 0,C 180,E1 -27845.772,E2 -27845.772} C_VEL
LIN {X 0,Y 87.953,Z 698.06,A -85,B 0,C 180,E1 -27854.276,E2 -27854.276} C_VEL
LIN {X 0,Y 89.641,Z 696.639,A -85,B 0,C 180,E1 -27856.421,E2 -27856.421} C_VEL
LIN {X 0,Y 93.117,Z 694.375,A -85,B 0,C 180,E1 -27859.004,E2 -27859.004} C_VEL
LIN {X 0,Y 91.623,Z 693.445,A -85,B 0,C 180,E1 -27862.147,E2 -27862.147} C_VEL
LIN {X 0,Y 82.969,Z 692.197,A -85,B 0,C 180,E1 -27874.943,E2 -27874.943} C_VEL
LIN {X 0,Y 84.613,Z 687.996,A -85,B 0,C 180,E1 -27909.563,E2 -27909.563} C_VEL
LIN {X 0,Y 101.842,Z 684.785,A -85,B 0,C 180,E1 -27928.886,E2 -27928.886} C_VEL
LIN {X 0,Y 106.578,Z 683.938,A -85,B 0,C 180,E1 -27931.84,E2 -27931.84} C_VEL
LIN {X 0,Y 105.169,Z 685.81,A -85,B 0,C 180,E1 -27933.756,E2 -27933.756} C_VEL
LIN {X 0,Y 95.366,Z 693.012,A -85,B 0,C 180,E1 -27939.303,E2 -27939.303} C_VEL
LIN {X 0,Y 86.535,Z 698.912,A -85,B 0,C 180,E1 -27946.342,E2 -27946.342} C_VEL
LIN {X 0,Y 80.895,Z 702.399,A -85,B 0,C 180,E1 -27952.543,E2 -27952.543} C_VEL
LIN {X 0,Y 74.867,Z 705.951,A -85,B 0,C 180,E1 -27962.006,E2 -27962.006} C_VEL
LIN {X 0,Y 71.097,Z 708.292,A -85,B 0,C 180,E1 -27972.748,E2 -27972.748} C_VEL
LIN {X 0,Y 69.548,Z 709.477,A -85,B 0,C 180,E1 -27984.199,E2 -27984.199} C_VEL
LIN {X 0,Y 69.573,Z 709.634,A -85,B 0,C 180,E1 -27989.999,E2 -27989.999} C_VEL
LIN {X 0,Y 70.046,Z 709.051,A -85,B 0,C 180,E1 -28001.575,E2 -28001.575} C_VEL
LIN {X 0,Y 72.652,Z 707.325,A -85,B 0,C 180,E1 -28012.764,E2 -28012.764} C_VEL
LIN {X 0,Y 77.602,Z 704.426,A -85,B 0,C 180,E1 -28022.914,E2 -28022.914} C_VEL
LIN {X 0,Y 84.432,Z 700.283,A -85,B 0,C 180,E1 -28031.751,E2 -28031.751} C_VEL
LIN {X 0,Y 92.969,Z 694.785,A -85,B 0,C 180,E1 -28039.107,E2 -28039.107} C_VEL
LIN {X 0,Y 102.788,Z 687.783,A -85,B 0,C 180,E1 -28045.132,E2 -28045.132} C_VEL
LIN {X 0,Y 111.981,Z 680.315,A -85,B 0,C 180,E1 -28049.602,E2 -28049.602} C_VEL
LIN {X 0,Y 121.871,Z 671.244,A -85,B 0,C 180,E1 -28053.36,E2 -28053.36} C_VEL
LIN {X 0,Y 130.719,Z 662.015,A -85,B 0,C 180,E1 -28056.062,E2 -28056.062} C_VEL
LIN {X 0,Y 140.567,Z 650.111,A -85,B 0,C 180,E1 -28058.622,E2 -28058.622} C_VEL
LIN {X 0,Y 149.092,Z 637.955,A -85,B 0,C 180,E1 -28060.522,E2 -28060.522} C_VEL
LIN {X 0,Y 156.931,Z 624.551,A -85,B 0,C 180,E1 -28062.112,E2 -28062.112} C_VEL
LIN {X 0,Y 163.293,Z 611.421,A -85,B 0,C 180,E1 -28063.259,E2 -28063.259} C_VEL
LIN {X 0,Y 168.938,Z 597.017,A -85,B 0,C 180,E1 -28064.159,E2 -28064.159} C_VEL
LIN {X 0,Y 173.405,Z 582.079,A -85,B 0,C 180,E1 -28064.819,E2 -28064.819} C_VEL
LIN {X 0,Y 176.64,Z 566.467,A -85,B 0,C 180,E1 -28065.307,E2 -28065.307} C_VEL
LIN {X 0,Y 181.137,Z 527.853,A -85,B 0,C 180,E1 -28066.136,E2 -28066.136} C_VEL
LIN {X 0,Y 182.087,Z 518.948,A -85,B 0,C 180,E1 -28066.362,E2 -28066.362} C_VEL
LIN {X 0,Y 180.857,Z 514.359,A -85,B 0,C 180,E1 -28068.938,E2 -28068.938} C_VEL
LIN {X 0,Y 179.57,Z 510.059,A -85,B 0,C 180,E1 -28072.409,E2 -28072.409} C_VEL
LIN {X 0,Y 178.769,Z 507.233,A -85,B 0,C 180,E1 -28075.914,E2 -28075.914} C_VEL
LIN {X 0,Y 178.486,Z 505.554,A -85,B 0,C 180,E1 -28080,E2 -28080} C_VEL
LIN {X 0,Y 178.563,Z 505.889,A -85,B 0,C 180,E1 -28082.255,E2 -28082.255} C_VEL
LIN {X 0,Y 179.507,Z 508.633,A -85,B 0,C 180,E1 -28087.31,E2 -28087.31} C_VEL
LIN {X 0,Y 180.756,Z 512.11,A -85,B 0,C 180,E1 -28090.732,E2 -28090.732} C_VEL
LIN {X 0,Y 182.202,Z 516.422,A -85,B 0,C 180,E1 -28093.67,E2 -28093.67} C_VEL
LIN {X 0,Y 176.586,Z 565.709,A -85,B 0,C 180,E1 -28094.757,E2 -28094.757} C_VEL
LIN {X 0,Y 173.853,Z 579.441,A -85,B 0,C 180,E1 -28095.172,E2 -28095.172} C_VEL
LIN {X 0,Y 169.788,Z 593.849,A -85,B 0,C 180,E1 -28095.766,E2 -28095.766} C_VEL
LIN {X 0,Y 164.948,Z 607.024,A -85,B 0,C 180,E1 -28096.532,E2 -28096.532} C_VEL
LIN {X 0,Y 158.542,Z 620.983,A -85,B 0,C 180,E1 -28097.624,E2 -28097.624} C_VEL
LIN {X 0,Y 150.848,Z 634.776,A -85,B 0,C 180,E1 -28099.17,E2 -28099.17} C_VEL
LIN {X 0,Y 142.921,Z 646.591,A -85,B 0,C 180,E1 -28100.884,E2 -28100.884} C_VEL
LIN {X 0,Y 133.733,Z 658.214,A -85,B 0,C 180,E1 -28103.123,E2 -28103.123} C_VEL
LIN {X 0,Y 124.829,Z 667.991,A -85,B 0,C 180,E1 -28105.735,E2 -28105.735} C_VEL
LIN {X 0,Y 114.615,Z 677.67,A -85,B 0,C 180,E1 -28109.281,E2 -28109.281} C_VEL
LIN {X 0,Y 105.408,Z 685.497,A -85,B 0,C 180,E1 -28113.548,E2 -28113.548} C_VEL
LIN {X 0,Y 95.337,Z 692.904,A -85,B 0,C 180,E1 -28119.284,E2 -28119.284} C_VEL
LIN {X 0,Y 86.452,Z 698.776,A -85,B 0,C 180,E1 -28126.292,E2 -28126.292} C_VEL
LIN {X 0,Y 80.827,Z 702.243,A -85,B 0,C 180,E1 -28132.508,E2 -28132.508} C_VEL
LIN {X 0,Y 74.842,Z 705.755,A -85,B 0,C 180,E1 -28141.997,E2 -28141.997} C_VEL
LIN {X 0,Y 71.094,Z 708.062,A -85,B 0,C 180,E1 -28152.749,E2 -28152.749} C_VEL
LIN {X 0,Y 69.574,Z 709.217,A -85,B 0,C 180,E1 -28164.203,E2 -28164.203} C_VEL
LIN {X 0,Y 69.576,Z 709.365,A -85,B 0,C 180,E1 -28170.001,E2 -28170.001} C_VEL
LIN {X 0,Y 70.049,Z 708.765,A -85,B 0,C 180,E1 -28181.576,E2 -28181.576} C_VEL
LIN {X 0,Y 72.656,Z 707.015,A -85,B 0,C 180,E1 -28192.764,E2 -28192.764} C_VEL
LIN {X 0,Y 77.602,Z 704.084,A -85,B 0,C 180,E1 -28202.916,E2 -28202.916} C_VEL
LIN {X 0,Y 84.474,Z 699.905,A -85,B 0,C 180,E1 -28211.728,E2 -28211.728} C_VEL
LIN {X 0,Y 89.641,Z 696.639,A -85,B 0,C 180,E1 -28216.421,E2 -28216.421} C_VEL
LIN {X 0,Y 90.16,Z 695.939,A -85,B 0,C 180,E1 -28217.704,E2 -28217.704} C_VEL
LIN {X 0,Y 89.632,Z 695.509,A -85,B 0,C 180,E1 -28219.123,E2 -28219.123} C_VEL
LIN {X 0,Y 87.281,Z 695.263,A -85,B 0,C 180,E1 -28221.617,E2 -28221.617} C_VEL
LIN {X 0,Y 80.136,Z 695.625,A -85,B 0,C 180,E1 -28227.461,E2 -28227.461} C_VEL
LIN {X 0,Y 79.05,Z 695.539,A -85,B 0,C 180,E1 -28229.003,E2 -28229.003} C_VEL
LIN {X 0,Y 73.501,Z 693.618,A -85,B 0,C 180,E1 -28248.976,E2 -28248.976} C_VEL
LIN {X 0,Y 78.333,Z 691.329,A -85,B 0,C 180,E1 -28270.338,E2 -28270.338} C_VEL
LIN {X 0,Y 97.427,Z 688.22,A -85,B 0,C 180,E1 -28291.385,E2 -28291.385} C_VEL
LIN {X 0,Y 95.645,Z 689.858,A -85,B 0,C 180,E1 -28293.134,E2 -28293.134} C_VEL
LIN {X 0,Y 86.096,Z 696.129,A -85,B 0,C 180,E1 -28299.15,E2 -28299.15} C_VEL
LIN {X 0,Y 78.505,Z 700.635,A -85,B 0,C 180,E1 -28305.741,E2 -28305.741} C_VEL
LIN {X 0,Y 71.745,Z 704.317,A -85,B 0,C 180,E1 -28314.001,E2 -28314.001} C_VEL
LIN {X 0,Y 66.124,Z 707.256,A -85,B 0,C 180,E1 -28324.84,E2 -28324.84} C_VEL
LIN {X 0,Y 63.095,Z 709.014,A -85,B 0,C 180,E1 -28337.127,E2 -28337.127} C_VEL
LIN {X 0,Y 62.49,Z 709.62,A -85,B 0,C 180,E1 -28349.999,E2 -28349.999} C_VEL
LIN {X 0,Y 63.091,Z 709.037,A -85,B 0,C 180,E1 -28362.872,E2 -28362.872} C_VEL
LIN {X 0,Y 66.111,Z 707.311,A -85,B 0,C 180,E1 -28375.164,E2 -28375.164} C_VEL
LIN {X 0,Y 71.686,Z 704.411,A -85,B 0,C 180,E1 -28386.031,E2 -28386.031} C_VEL
LIN {X 0,Y 79.232,Z 700.267,A -85,B 0,C 180,E1 -28395.203,E2 -28395.203} C_VEL
LIN {X 0,Y 88.458,Z 694.768,A -85,B 0,C 180,E1 -28402.607,E2 -28402.607} C_VEL
LIN {X 0,Y 96.152,Z 689.67,A -85,B 0,C 180,E1 -28407.199,E2 -28407.199} C_VEL
LIN {X 0,Y 105.752,Z 682.53,A -85,B 0,C 180,E1 -28411.709,E2 -28411.709} C_VEL
LIN {X 0,Y 115.844,Z 673.945,A -85,B 0,C 180,E1 -28415.507,E2 -28415.507} C_VEL
LIN {X 0,Y 126.45,Z 663.605,A -85,B 0,C 180,E1 -28418.582,E2 -28418.582} C_VEL
LIN {X 0,Y 135.76,Z 652.99,A -85,B 0,C 180,E1 -28420.867,E2 -28420.867} C_VEL
LIN {X 0,Y 144.487,Z 641.411,A -85,B 0,C 180,E1 -28422.665,E2 -28422.665} C_VEL
LIN {X 0,Y 152.454,Z 628.795,A -85,B 0,C 180,E1 -28424.2,E2 -28424.2} C_VEL
LIN {X 0,Y 159.76,Z 614.853,A -85,B 0,C 180,E1 -28425.42,E2 -28425.42} C_VEL
LIN {X 0,Y 165.909,Z 600.282,A -85,B 0,C 180,E1 -28426.322,E2 -28426.322} C_VEL
LIN {X 0,Y 170.854,Z 584.987,A -85,B 0,C 180,E1 -28427,E2 -28427} C_VEL
LIN {X 0,Y 174.29,Z 570.059,A -85,B 0,C 180,E1 -28427.468,E2 -28427.468} C_VEL
LIN {X 0,Y 176.731,Z 552.751,A -85,B 0,C 180,E1 -28427.869,E2 -28427.869} C_VEL
LIN {X 0,Y 180.087,Z 523.059,A -85,B 0,C 180,E1 -28428.434,E2 -28428.434} C_VEL
LIN {X 0,Y 179.101,Z 519.229,A -85,B 0,C 180,E1 -28430.969,E2 -28430.969} C_VEL
LIN {X 0,Y 178.172,Z 515.576,A -85,B 0,C 180,E1 -28434.34,E2 -28434.34} C_VEL
LIN {X 0,Y 177.787,Z 514.027,A -85,B 0,C 180,E1 -28436.6,E2 -28436.6} C_VEL
LIN {X 0,Y 177.617,Z 512.628,A -85,B 0,C 180,E1 -28440,E2 -28440} C_VEL
LIN {X 0,Y 177.675,Z 512.883,A -85,B 0,C 180,E1 -28441.983,E2 -28441.983} C_VEL
LIN {X 0,Y 178.463,Z 515.467,A -85,B 0,C 180,E1 -28446.785,E2 -28446.785} C_VEL
LIN {X 0,Y 179.551,Z 518.812,A -85,B 0,C 180,E1 -28450.085,E2 -28450.085} C_VEL
LIN {X 0,Y 180.177,Z 520.85,A -85,B 0,C 180,E1 -28451.572,E2 -28451.572} C_VEL
LIN {X 0,Y 174.881,Z 566.052,A -85,B 0,C 180,E1 -28452.515,E2 -28452.515} C_VEL
LIN {X 0,Y 172.133,Z 579.514,A -85,B 0,C 180,E1 -28452.894,E2 -28452.894} C_VEL
LIN {X 0,Y 168.003,Z 593.902,A -85,B 0,C 180,E1 -28453.442,E2 -28453.442} C_VEL
LIN {X 0,Y 163.069,Z 607.066,A -85,B 0,C 180,E1 -28454.138,E2 -28454.138} C_VEL
LIN {X 0,Y 156.536,Z 621.017,A -85,B 0,C 180,E1 -28455.142,E2 -28455.142} C_VEL
LIN {X 0,Y 148.657,Z 634.806,A -85,B 0,C 180,E1 -28456.571,E2 -28456.571} C_VEL
LIN {X 0,Y 140.546,Z 646.617,A -85,B 0,C 180,E1 -28458.178,E2 -28458.178} C_VEL
LIN {X 0,Y 131.093,Z 658.237,A -85,B 0,C 180,E1 -28460.251,E2 -28460.251} C_VEL
LIN {X 0,Y 121.897,Z 668.011,A -85,B 0,C 180,E1 -28462.709,E2 -28462.709} C_VEL
LIN {X 0,Y 111.445,Z 677.566,A -85,B 0,C 180,E1 -28466.021,E2 -28466.021} C_VEL
LIN {X 0,Y 101.636,Z 685.514,A -85,B 0,C 180,E1 -28470.191,E2 -28470.191} C_VEL
LIN {X 0,Y 90.965,Z 692.921,A -85,B 0,C 180,E1 -28475.785,E2 -28475.785} C_VEL
LIN {X 0,Y 81.425,Z 698.792,A -85,B 0,C 180,E1 -28482.807,E2 -28482.807} C_VEL
LIN {X 0,Y 75.277,Z 702.258,A -85,B 0,C 180,E1 -28489.192,E2 -28489.192} C_VEL
LIN {X 0,Y 68.625,Z 705.769,A -85,B 0,C 180,E1 -28499.2,E2 -28499.2} C_VEL
LIN {X 0,Y 64.295,Z 708.076,A -85,B 0,C 180,E1 -28510.858,E2 -28510.858} C_VEL
LIN {X 0,Y 62.514,Z 709.23,A -85,B 0,C 180,E1 -28523.546,E2 -28523.546} C_VEL
LIN {X 0,Y 62.493,Z 709.379,A -85,B 0,C 180,E1 -28530.001,E2 -28530.001} C_VEL
LIN {X 0,Y 63.094,Z 708.779,A -85,B 0,C 180,E1 -28542.873,E2 -28542.873} C_VEL
LIN {X 0,Y 66.115,Z 707.029,A -85,B 0,C 180,E1 -28555.164,E2 -28555.164} C_VEL
LIN {X 0,Y 71.69,Z 704.098,A -85,B 0,C 180,E1 -28566.03,E2 -28566.03} C_VEL
LIN {X 0,Y 79.276,Z 699.918,A -85,B 0,C 180,E1 -28575.172,E2 -28575.172} C_VEL
LIN {X 0,Y 85.245,Z 696.44,A -85,B 0,C 180,E1 -28580.175,E2 -28580.175} C_VEL
LIN {X 0,Y 84.282,Z 696.11,A -85,B 0,C 180,E1 -28581.875,E2 -28581.875} C_VEL
LIN {X 0,Y 79.05,Z 695.539,A -85,B 0,C 180,E1 -28589.003,E2 -28589.003} C_VEL
LIN {X 0,Y 76.447,Z 695.43,A -85,B 0,C 180,E1 -28592.913,E2 -28592.913} C_VEL
LIN {X 0,Y 67.694,Z 696.312,A -85,B 0,C 180,E1 -28607.086,E2 -28607.086} C_VEL
LIN {X 0,Y 67.108,Z 696.127,A -85,B 0,C 180,E1 -28612.063,E2 -28612.063} C_VEL
LIN {X 0,Y 74.703,Z 693.904,A -85,B 0,C 180,E1 -28636.394,E2 -28636.394} C_VEL
LIN {X 0,Y 87.513,Z 692.169,A -85,B 0,C 180,E1 -28650.336,E2 -28650.336} C_VEL
LIN {X 0,Y 86.175,Z 693.471,A -85,B 0,C 180,E1 -28652.444,E2 -28652.444} C_VEL
LIN {X 0,Y 76.811,Z 698.885,A -85,B 0,C 180,E1 -28658.946,E2 -28658.946} C_VEL
LIN {X 0,Y 70.077,Z 702.372,A -85,B 0,C 180,E1 -28665.409,E2 -28665.409} C_VEL
LIN {X 0,Y 62.61,Z 705.924,A -85,B 0,C 180,E1 -28675.857,E2 -28675.857} C_VEL
LIN {X 0,Y 57.59,Z 708.265,A -85,B 0,C 180,E1 -28688.524,E2 -28688.524} C_VEL
LIN {X 0,Y 55.404,Z 709.45,A -85,B 0,C 180,E1 -28702.711,E2 -28702.711} C_VEL
LIN {X 0,Y 55.39,Z 709.606,A -85,B 0,C 180,E1 -28709.999,E2 -28709.999} C_VEL
LIN {X 0,Y 56.153,Z 709.023,A -85,B 0,C 180,E1 -28724.495,E2 -28724.495} C_VEL
LIN {X 0,Y 59.713,Z 707.296,A -85,B 0,C 180,E1 -28738.084,E2 -28738.084} C_VEL
LIN {X 0,Y 66.018,Z 704.396,A -85,B 0,C 180,E1 -28749.697,E2 -28749.697} C_VEL
LIN {X 0,Y 74.358,Z 700.251,A -85,B 0,C 180,E1 -28759.123,E2 -28759.123} C_VEL
LIN {X 0,Y 84.293,Z 694.752,A -85,B 0,C 180,E1 -28766.486,E2 -28766.486} C_VEL
LIN {X 0,Y 95.339,Z 687.748,A -85,B 0,C 180,E1 -28772.2,E2 -28772.2} C_VEL
LIN {X 0,Y 105.034,Z 680.635,A -85,B 0,C 180,E1 -28776.16,E2 -28776.16} C_VEL
LIN {X 0,Y 116.17,Z 671.204,A -85,B 0,C 180,E1 -28779.67,E2 -28779.67} C_VEL
LIN {X 0,Y 125.61,Z 661.972,A -85,B 0,C 180,E1 -28782.019,E2 -28782.019} C_VEL
LIN {X 0,Y 135.221,Z 651.037,A -85,B 0,C 180,E1 -28784.053,E2 -28784.053} C_VEL
LIN {X 0,Y 144.154,Z 639.068,A -85,B 0,C 180,E1 -28785.689,E2 -28785.689} C_VEL
LIN {X 0,Y 152.337,Z 625.929,A -85,B 0,C 180,E1 -28787.055,E2 -28787.055} C_VEL
LIN {X 0,Y 158.952,Z 613.084,A -85,B 0,C 180,E1 -28788.027,E2 -28788.027} C_VEL
LIN {X 0,Y 164.788,Z 599.135,A -85,B 0,C 180,E1 -28788.789,E2 -28788.789} C_VEL
LIN {X 0,Y 169.61,Z 584.188,A -85,B 0,C 180,E1 -28789.362,E2 -28789.362} C_VEL
LIN {X 0,Y 173.002,Z 569.397,A -85,B 0,C 180,E1 -28789.772,E2 -28789.772} C_VEL
LIN {X 0,Y 175.58,Z 550.754,A -85,B 0,C 180,E1 -28790.188,E2 -28790.188} C_VEL
LIN {X 0,Y 178.277,Z 527.315,A -85,B 0,C 180,E1 -28790.613,E2 -28790.613} C_VEL
LIN {X 0,Y 177.311,Z 522.986,A -85,B 0,C 180,E1 -28794.17,E2 -28794.17} C_VEL
LIN {X 0,Y 176.876,Z 520.993,A -85,B 0,C 180,E1 -28796.898,E2 -28796.898} C_VEL
LIN {X 0,Y 176.743,Z 519.75,A -85,B 0,C 180,E1 -28800,E2 -28800} C_VEL
LIN {X 0,Y 176.791,Z 519.875,A -85,B 0,C 180,E1 -28801.708,E2 -28801.708} C_VEL
LIN {X 0,Y 177.435,Z 522.299,A -85,B 0,C 180,E1 -28806.253,E2 -28806.253} C_VEL
LIN {X 0,Y 178.359,Z 525.496,A -85,B 0,C 180,E1 -28809.403,E2 -28809.403} C_VEL
LIN {X 0,Y 173.492,Z 566.094,A -85,B 0,C 180,E1 -28810.224,E2 -28810.224} C_VEL
LIN {X 0,Y 170.484,Z 580.466,A -85,B 0,C 180,E1 -28810.602,E2 -28810.602} C_VEL
LIN {X 0,Y 166.079,Z 595.219,A -85,B 0,C 180,E1 -28811.12,E2 -28811.12} C_VEL
LIN {X 0,Y 160.65,Z 609.054,A -85,B 0,C 180,E1 -28811.807,E2 -28811.807} C_VEL
LIN {X 0,Y 154.008,Z 622.609,A -85,B 0,C 180,E1 -28812.729,E2 -28812.729} C_VEL
LIN {X 0,Y 146.345,Z 635.52,A -85,B 0,C 180,E1 -28813.978,E2 -28813.978} C_VEL
LIN {X 0,Y 137.674,Z 647.699,A -85,B 0,C 180,E1 -28815.523,E2 -28815.523} C_VEL
LIN {X 0,Y 128.8,Z 658.26,A -85,B 0,C 180,E1 -28817.276,E2 -28817.276} C_VEL
LIN {X 0,Y 119.328,Z 668.032,A -85,B 0,C 180,E1 -28819.552,E2 -28819.552} C_VEL
LIN {X 0,Y 108.499,Z 677.585,A -85,B 0,C 180,E1 -28822.626,E2 -28822.626} C_VEL
LIN {X 0,Y 99.698,Z 684.505,A -85,B 0,C 180,E1 -28826.002,E2 -28826.002} C_VEL
LIN {X 0,Y 89.688,Z 691.234,A -85,B 0,C 180,E1 -28830.463,E2 -28830.463} C_VEL
LIN {X 0,Y 79.189,Z 697.467,A -85,B 0,C 180,E1 -28836.99,E2 -28836.99} C_VEL
LIN {X 0,Y 70.004,Z 702.273,A -85,B 0,C 180,E1 -28845.352,E2 -28845.352} C_VEL
LIN {X 0,Y 62.581,Z 705.784,A -85,B 0,C 180,E1 -28855.84,E2 -28855.84} C_VEL
LIN {X 0,Y 57.586,Z 708.09,A -85,B 0,C 180,E1 -28868.524,E2 -28868.524} C_VEL
LIN {X 0,Y 55.454,Z 709.244,A -85,B 0,C 180,E1 -28882.72,E2 -28882.72} C_VEL
LIN {X 0,Y 55.394,Z 709.393,A -85,B 0,C 180,E1 -28890.001,E2 -28890.001} C_VEL
LIN {X 0,Y 56.155,Z 708.792,A -85,B 0,C 180,E1 -28904.497,E2 -28904.497} C_VEL
LIN {X 0,Y 59.717,Z 707.042,A -85,B 0,C 180,E1 -28918.084,E2 -28918.084} C_VEL
LIN {X 0,Y 66.03,Z 704.112,A -85,B 0,C 180,E1 -28929.69,E2 -28929.69} C_VEL
LIN {X 0,Y 74.401,Z 699.932,A -85,B 0,C 180,E1 -28939.086,E2 -28939.086} C_VEL
LIN {X 0,Y 75.817,Z 699.189,A -85,B 0,C 180,E1 -28940.314,E2 -28940.314} C_VEL
LIN {X 0,Y 76.405,Z 698.508,A -85,B 0,C 180,E1 -28942.103,E2 -28942.103} C_VEL
LIN {X 0,Y 67.681,Z 696.969,A -85,B 0,C 180,E1 -28961.85,E2 -28961.85} C_VEL
LIN {X 0,Y 67.108,Z 696.127,A -85,B 0,C 180,E1 -28972.063,E2 -28972.063} C_VEL
LIN {X 0,Y 67.035,Z 695.944,A -85,B 0,C 180,E1 -28977.107,E2 -28977.107} C_VEL
LIN {X 0,Y 66.294,Z 696.354,A -85,B 0,C 180,E1 -28985.613,E2 -28985.613} C_VEL
LIN {X 0,Y 66.586,Z 696.756,A -85,B 0,C 180,E1 -28992.482,E2 -28992.482} C_VEL
LIN {X 0,Y 68.114,Z 696.768,A -85,B 0,C 180,E1 -28997.361,E2 -28997.361} C_VEL
LIN {X 0,Y 68.956,Z 696.674,A -85,B 0,C 180,E1 -28998.855,E2 -28998.855} C_VEL
LIN {X 0,Y 78.467,Z 695.569,A -85,B 0,C 180,E1 -29009.832,E2 -29009.832} C_VEL
LIN {X 0,Y 76.912,Z 696.584,A -85,B 0,C 180,E1 -29011.519,E2 -29011.519} C_VEL
LIN {X 0,Y 67.674,Z 701.234,A -85,B 0,C 180,E1 -29018.544,E2 -29018.544} C_VEL
LIN {X 0,Y 60.741,Z 704.29,A -85,B 0,C 180,E1 -29026.033,E2 -29026.033} C_VEL
LIN {X 0,Y 53.523,Z 707.228,A -85,B 0,C 180,E1 -29038.315,E2 -29038.315} C_VEL
LIN {X 0,Y 49.286,Z 708.986,A -85,B 0,C 180,E1 -29053.428,E2 -29053.428} C_VEL
LIN {X 0,Y 48.305,Z 709.593,A -85,B 0,C 180,E1 -29069.999,E2 -29069.999} C_VEL
LIN {X 0,Y 49.282,Z 709.009,A -85,B 0,C 180,E1 -29086.571,E2 -29086.571} C_VEL
LIN {X 0,Y 53.507,Z 707.282,A -85,B 0,C 180,E1 -29101.694,E2 -29101.694} C_VEL
LIN {X 0,Y 60.671,Z 704.381,A -85,B 0,C 180,E1 -29114.028,E2 -29114.028} C_VEL
LIN {X 0,Y 69.889,Z 700.236,A -85,B 0,C 180,E1 -29123.558,E2 -29123.558} C_VEL
LIN {X 0,Y 80.558,Z 694.735,A -85,B 0,C 180,E1 -29130.74,E2 -29130.74} C_VEL
LIN {X 0,Y 92.221,Z 687.73,A -85,B 0,C 180,E1 -29136.134,E2 -29136.134} C_VEL
LIN {X 0,Y 103.005,Z 680.094,A -85,B 0,C 180,E1 -29140.053,E2 -29140.053} C_VEL
LIN {X 0,Y 113.889,Z 671.184,A -85,B 0,C 180,E1 -29143.035,E2 -29143.035} C_VEL
LIN {X 0,Y 123.592,Z 661.95,A -85,B 0,C 180,E1 -29145.17,E2 -29145.17} C_VEL
LIN {X 0,Y 133.444,Z 651.013,A -85,B 0,C 180,E1 -29146.988,E2 -29146.988} C_VEL
LIN {X 0,Y 142.768,Z 638.745,A -85,B 0,C 180,E1 -29148.505,E2 -29148.505} C_VEL
LIN {X 0,Y 150.903,Z 625.897,A -85,B 0,C 180,E1 -29149.688,E2 -29149.688} C_VEL
LIN {X 0,Y 157.633,Z 613.046,A -85,B 0,C 180,E1 -29150.551,E2 -29150.551} C_VEL
LIN {X 0,Y 163.556,Z 599.088,A -85,B 0,C 180,E1 -29151.228,E2 -29151.228} C_VEL
LIN {X 0,Y 168.445,Z 584.126,A -85,B 0,C 180,E1 -29151.733,E2 -29151.733} C_VEL
LIN {X 0,Y 171.936,Z 569.028,A -85,B 0,C 180,E1 -29152.112,E2 -29152.112} C_VEL
LIN {X 0,Y 174.503,Z 550.691,A -85,B 0,C 180,E1 -29152.48,E2 -29152.48} C_VEL
LIN {X 0,Y 176.691,Z 532.02,A -85,B 0,C 180,E1 -29152.791,E2 -29152.791} C_VEL
LIN {X 0,Y 176.131,Z 528.993,A -85,B 0,C 180,E1 -29155.737,E2 -29155.737} C_VEL
LIN {X 0,Y 175.89,Z 527.578,A -85,B 0,C 180,E1 -29158.139,E2 -29158.139} C_VEL
LIN {X 0,Y 175.872,Z 526.84,A -85,B 0,C 180,E1 -29160,E2 -29160} C_VEL
LIN {X 0,Y 175.92,Z 526.977,A -85,B 0,C 180,E1 -29161.717,E2 -29161.717} C_VEL
LIN {X 0,Y 176.45,Z 529.259,A -85,B 0,C 180,E1 -29165.858,E2 -29165.858} C_VEL
LIN {X 0,Y 176.784,Z 530.54,A -85,B 0,C 180,E1 -29167.277,E2 -29167.277} C_VEL
LIN {X 0,Y 172.414,Z 565.942,A -85,B 0,C 180,E1 -29167.899,E2 -29167.899} C_VEL
LIN {X 0,Y 169.32,Z 580.536,A -85,B 0,C 180,E1 -29168.238,E2 -29168.238} C_VEL
LIN {X 0,Y 164.861,Z 595.27,A -85,B 0,C 180,E1 -29168.706,E2 -29168.706} C_VEL
LIN {X 0,Y 159.351,Z 609.095,A -85,B 0,C 180,E1 -29169.312,E2 -29169.312} C_VEL
LIN {X 0,Y 152.599,Z 622.642,A -85,B 0,C 180,E1 -29170.124,E2 -29170.124} C_VEL
LIN {X 0,Y 144.422,Z 636.116,A -85,B 0,C 180,E1 -29171.304,E2 -29171.304} C_VEL
LIN {X 0,Y 135.946,Z 647.724,A -85,B 0,C 180,E1 -29172.637,E2 -29172.637} C_VEL
LIN {X 0,Y 126.866,Z 658.283,A -85,B 0,C 180,E1 -29174.2,E2 -29174.2} C_VEL
LIN {X 0,Y 117.138,Z 668.053,A -85,B 0,C 180,E1 -29176.269,E2 -29176.269} C_VEL
LIN {X 0,Y 105.961,Z 677.604,A -85,B 0,C 180,E1 -29179.067,E2 -29179.067} C_VEL
LIN {X 0,Y 96.767,Z 684.523,A -85,B 0,C 180,E1 -29182.18,E2 -29182.18} C_VEL
LIN {X 0,Y 86.283,Z 691.251,A -85,B 0,C 180,E1 -29186.366,E2 -29186.366} C_VEL
LIN {X 0,Y 75.096,Z 697.483,A -85,B 0,C 180,E1 -29192.619,E2 -29192.619} C_VEL
LIN {X 0,Y 65.101,Z 702.288,A -85,B 0,C 180,E1 -29200.915,E2 -29200.915} C_VEL
LIN {X 0,Y 56.802,Z 705.799,A -85,B 0,C 180,E1 -29211.784,E2 -29211.784} C_VEL
LIN {X 0,Y 51.007,Z 708.105,A -85,B 0,C 180,E1 -29225.585,E2 -29225.585} C_VEL
LIN {X 0,Y 48.4,Z 709.258,A -85,B 0,C 180,E1 -29241.652,E2 -29241.652} C_VEL
LIN {X 0,Y 48.309,Z 709.406,A -85,B 0,C 180,E1 -29250.001,E2 -29250.001} C_VEL
LIN {X 0,Y 49.285,Z 708.806,A -85,B 0,C 180,E1 -29266.572,E2 -29266.572} C_VEL
LIN {X 0,Y 53.511,Z 707.056,A -85,B 0,C 180,E1 -29281.693,E2 -29281.693} C_VEL
LIN {X 0,Y 60.688,Z 704.125,A -85,B 0,C 180,E1 -29294.015,E2 -29294.015} C_VEL
LIN {X 0,Y 66.84,Z 701.395,A -85,B 0,C 180,E1 -29300.886,E2 -29300.886} C_VEL
LIN {X 0,Y 67.767,Z 700.588,A -85,B 0,C 180,E1 -29303.394,E2 -29303.394} C_VEL
LIN {X 0,Y 60.57,Z 698.631,A -85,B 0,C 180,E1 -29333.338,E2 -29333.338} C_VEL
LIN {X 0,Y 68.956,Z 696.674,A -85,B 0,C 180,E1 -29358.855,E2 -29358.855} C_VEL
LIN {X 0,Y 69.665,Z 696.761,A -85,B 0,C 180,E1 -29360.92,E2 -29360.92} C_VEL
LIN {X 0,Y 69.463,Z 697.356,A -85,B 0,C 180,E1 -29363.621,E2 -29363.621} C_VEL
LIN {X 0,Y 67.909,Z 698.639,A -85,B 0,C 180,E1 -29367.296,E2 -29367.296} C_VEL
LIN {X 0,Y 64.807,Z 700.45,A -85,B 0,C 180,E1 -29371.604,E2 -29371.604} C_VEL
LIN {X 0,Y 60.949,Z 702.244,A -85,B 0,C 180,E1 -29375.644,E2 -29375.644} C_VEL
LIN {X 0,Y 51.405,Z 705.897,A -85,B 0,C 180,E1 -29386.874,E2 -29386.874} C_VEL
LIN {X 0,Y 44.614,Z 708.238,A -85,B 0,C 180,E1 -29401.796,E2 -29401.796} C_VEL
LIN {X 0,Y 41.328,Z 709.423,A -85,B 0,C 180,E1 -29420.208,E2 -29420.208} C_VEL
LIN {X 0,Y 41.19,Z 709.579,A -85,B 0,C 180,E1 -29429.999,E2 -29429.999} C_VEL
LIN {X 0,Y 42.507,Z 708.995,A -85,B 0,C 180,E1 -29449.309,E2 -29449.309} C_VEL
LIN {X 0,Y 47.567,Z 707.268,A -85,B 0,C 180,E1 -29466.226,E2 -29466.226} C_VEL
LIN {X 0,Y 55.738,Z 704.366,A -85,B 0,C 180,E1 -29479.159,E2 -29479.159} C_VEL
LIN {X 0,Y 65.898,Z 700.22,A -85,B 0,C 180,E1 -29488.56,E2 -29488.56} C_VEL
LIN {X 0,Y 77.312,Z 694.719,A -85,B 0,C 180,E1 -29495.372,E2 -29495.372} C_VEL
LIN {X 0,Y 89.57,Z 687.713,A -85,B 0,C 180,E1 -29500.314,E2 -29500.314} C_VEL
LIN {X 0,Y 100.124,Z 680.581,A -85,B 0,C 180,E1 -29503.693,E2 -29503.693} C_VEL
LIN {X 0,Y 112.017,Z 671.163,A -85,B 0,C 180,E1 -29506.525,E2 -29506.525} C_VEL
LIN {X 0,Y 121.96,Z 661.928,A -85,B 0,C 180,E1 -29508.414,E2 -29508.414} C_VEL
LIN {X 0,Y 132.865,Z 650.013,A -85,B 0,C 180,E1 -29510.123,E2 -29510.123} C_VEL
LIN {X 0,Y 142.145,Z 637.843,A -85,B 0,C 180,E1 -29511.433,E2 -29511.433} C_VEL
LIN {X 0,Y 150.647,Z 624.418,A -85,B 0,C 180,E1 -29512.46,E2 -29512.46} C_VEL
LIN {X 0,Y 157.482,Z 611.267,A -85,B 0,C 180,E1 -29513.195,E2 -29513.195} C_VEL
LIN {X 0,Y 163.485,Z 596.822,A -85,B 0,C 180,E1 -29513.777,E2 -29513.777} C_VEL
LIN {X 0,Y 168.219,Z 581.814,A -85,B 0,C 180,E1 -29514.187,E2 -29514.187} C_VEL
LIN {X 0,Y 171.534,Z 566.742,A -85,B 0,C 180,E1 -29514.506,E2 -29514.506} C_VEL
LIN {X 0,Y 175.328,Z 536.966,A -85,B 0,C 180,E1 -29515.03,E2 -29515.03} C_VEL
LIN {X 0,Y 175.05,Z 534.84,A -85,B 0,C 180,E1 -29517.699,E2 -29517.699} C_VEL
LIN {X 0,Y 175.002,Z 533.929,A -85,B 0,C 180,E1 -29520,E2 -29520} C_VEL
LIN {X 0,Y 175.048,Z 534.084,A -85,B 0,C 180,E1 -29521.725,E2 -29521.725} C_VEL
LIN {X 0,Y 175.404,Z 535.848,A -85,B 0,C 180,E1 -29525.04,E2 -29525.04} C_VEL
LIN {X 0,Y 171.536,Z 566.357,A -85,B 0,C 180,E1 -29525.557,E2 -29525.557} C_VEL
LIN {X 0,Y 168.451,Z 580.607,A -85,B 0,C 180,E1 -29525.851,E2 -29525.851} C_VEL
LIN {X 0,Y 163.936,Z 595.322,A -85,B 0,C 180,E1 -29526.251,E2 -29526.251} C_VEL
LIN {X 0,Y 158.358,Z 609.135,A -85,B 0,C 180,E1 -29526.779,E2 -29526.779} C_VEL
LIN {X 0,Y 151.51,Z 622.676,A -85,B 0,C 180,E1 -29527.474,E2 -29527.474} C_VEL
LIN {X 0,Y 143.653,Z 635.452,A -85,B 0,C 180,E1 -29528.439,E2 -29528.439} C_VEL
LIN {X 0,Y 134.569,Z 647.749,A -85,B 0,C 180,E1 -29529.681,E2 -29529.681} C_VEL
LIN {X 0,Y 125.31,Z 658.306,A -85,B 0,C 180,E1 -29531.044,E2 -29531.044} C_VEL
LIN {X 0,Y 115.345,Z 668.073,A -85,B 0,C 180,E1 -29532.87,E2 -29532.87} C_VEL
LIN {X 0,Y 103.852,Z 677.623,A -85,B 0,C 180,E1 -29535.349,E2 -29535.349} C_VEL
LIN {X 0,Y 95.839,Z 683.436,A -85,B 0,C 180,E1 -29537.579,E2 -29537.579} C_VEL
LIN {X 0,Y 86.456,Z 689.473,A -85,B 0,C 180,E1 -29540.799,E2 -29540.799} C_VEL
LIN {X 0,Y 74.386,Z 696.086,A -85,B 0,C 180,E1 -29546.162,E2 -29546.162} C_VEL
LIN {X 0,Y 65.915,Z 700.071,A -85,B 0,C 180,E1 -29551.464,E2 -29551.464} C_VEL
LIN {X 0,Y 55.763,Z 704.214,A -85,B 0,C 180,E1 -29560.871,E2 -29560.871} C_VEL
LIN {X 0,Y 47.57,Z 707.113,A -85,B 0,C 180,E1 -29573.776,E2 -29573.776} C_VEL
LIN {X 0,Y 42.508,Z 708.837,A -85,B 0,C 180,E1 -29590.692,E2 -29590.692} C_VEL
LIN {X 0,Y 41.197,Z 709.42,A -85,B 0,C 180,E1 -29610.001,E2 -29610.001} C_VEL
LIN {X 0,Y 42.509,Z 708.819,A -85,B 0,C 180,E1 -29629.31,E2 -29629.31} C_VEL
LIN {X 0,Y 47.572,Z 707.069,A -85,B 0,C 180,E1 -29646.225,E2 -29646.225} C_VEL
LIN {X 0,Y 55.76,Z 704.139,A -85,B 0,C 180,E1 -29659.135,E2 -29659.135} C_VEL
LIN {X 0,Y 59.78,Z 702.462,A -85,B 0,C 180,E1 -29663.999,E2 -29663.999} C_VEL
LIN {X 0,Y 54.68,Z 700.567,A -85,B 0,C 180,E1 -29700.001,E2 -29700.001} C_VEL
LIN {X 0,Y 68.641,Z 698.651,A -85,B 0,C 180,E1 -29728.501,E2 -29728.501} C_VEL
LIN {X 0,Y 67.46,Z 699.416,A -85,B 0,C 180,E1 -29730.466,E2 -29730.466} C_VEL
LIN {X 0,Y 60.949,Z 702.244,A -85,B 0,C 180,E1 -29735.644,E2 -29735.644} C_VEL
LIN {X 0,Y 56.533,Z 703.863,A -85,B 0,C 180,E1 -29739.132,E2 -29739.132} C_VEL
LIN {X 0,Y 48.377,Z 706.071,A -85,B 0,C 180,E1 -29744.801,E2 -29744.801} C_VEL
LIN {X 0,Y 42.111,Z 707.448,A -85,B 0,C 180,E1 -29750.786,E2 -29750.786} C_VEL
LIN {X 0,Y 38.386,Z 708.264,A -85,B 0,C 180,E1 -29757.257,E2 -29757.257} C_VEL
LIN {X 0,Y 37.488,Z 708.463,A -85,B 0,C 180,E1 -29759.894,E2 -29759.894} C_VEL
LIN {X 0,Y 34.344,Z 709.409,A -85,B 0,C 180,E1 -29778.19,E2 -29778.19} C_VEL
LIN {X 0,Y 34.083,Z 709.565,A -85,B 0,C 180,E1 -29789.998,E2 -29789.998} C_VEL
LIN {X 0,Y 35.845,Z 708.981,A -85,B 0,C 180,E1 -29813.086,E2 -29813.086} C_VEL
LIN {X 0,Y 42.011,Z 707.253,A -85,B 0,C 180,E1 -29832,E2 -29832} C_VEL
LIN {X 0,Y 51.337,Z 704.351,A -85,B 0,C 180,E1 -29845.224,E2 -29845.224} C_VEL
LIN {X 0,Y 62.465,Z 700.205,A -85,B 0,C 180,E1 -29854.168,E2 -29854.168} C_VEL
LIN {X 0,Y 74.617,Z 694.703,A -85,B 0,C 180,E1 -29860.367,E2 -29860.367} C_VEL
LIN {X 0,Y 87.425,Z 687.696,A -85,B 0,C 180,E1 -29864.721,E2 -29864.721} C_VEL
LIN {X 0,Y 99.065,Z 680.037,A -85,B 0,C 180,E1 -29867.871,E2 -29867.871} C_VEL
LIN {X 0,Y 110.574,Z 671.143,A -85,B 0,C 180,E1 -29870.118,E2 -29870.118} C_VEL
LIN {X 0,Y 120.73,Z 661.906,A -85,B 0,C 180,E1 -29871.732,E2 -29871.732} C_VEL
LIN {X 0,Y 131.829,Z 649.988,A -85,B 0,C 180,E1 -29873.179,E2 -29873.179} C_VEL
LIN {X 0,Y 141.26,Z 637.815,A -85,B 0,C 180,E1 -29874.289,E2 -29874.289} C_VEL
LIN {X 0,Y 149.88,Z 624.385,A -85,B 0,C 180,E1 -29875.152,E2 -29875.152} C_VEL
LIN {X 0,Y 156.799,Z 611.228,A -85,B 0,C 180,E1 -29875.77,E2 -29875.77} C_VEL
LIN {X 0,Y 162.822,Z 596.9,A -85,B 0,C 180,E1 -29876.256,E2 -29876.256} C_VEL
LIN {X 0,Y 167.638,Z 581.784,A -85,B 0,C 180,E1 -29876.607,E2 -29876.607} C_VEL
LIN {X 0,Y 171.106,Z 565.987,A -85,B 0,C 180,E1 -29876.88,E2 -29876.88} C_VEL
LIN {X 0,Y 174.194,Z 542.296,A -85,B 0,C 180,E1 -29877.272,E2 -29877.272} C_VEL
LIN {X 0,Y 174.13,Z 541.028,A -85,B 0,C 180,E1 -29880,E2 -29880} C_VEL
LIN {X 0,Y 174.169,Z 541.103,A -85,B 0,C 180,E1 -29881.517,E2 -29881.517} C_VEL
LIN {X 0,Y 174.234,Z 541.724,A -85,B 0,C 180,E1 -29882.828,E2 -29882.828} C_VEL
LIN {X 0,Y 170.929,Z 566.839,A -85,B 0,C 180,E1 -29883.199,E2 -29883.199} C_VEL
LIN {X 0,Y 167.903,Z 580.568,A -85,B 0,C 180,E1 -29883.441,E2 -29883.441} C_VEL
LIN {X 0,Y 163.25,Z 595.565,A -85,B 0,C 180,E1 -29883.783,E2 -29883.783} C_VEL
LIN {X 0,Y 157.677,Z 609.175,A -85,B 0,C 180,E1 -29884.213,E2 -29884.213} C_VEL
LIN {X 0,Y 150.751,Z 622.709,A -85,B 0,C 180,E1 -29884.798,E2 -29884.798} C_VEL
LIN {X 0,Y 142.995,Z 635.169,A -85,B 0,C 180,E1 -29885.6,E2 -29885.6} C_VEL
LIN {X 0,Y 134.417,Z 646.718,A -85,B 0,C 180,E1 -29886.58,E2 -29886.58} C_VEL
LIN {X 0,Y 124.14,Z 658.328,A -85,B 0,C 180,E1 -29887.808,E2 -29887.808} C_VEL
LIN {X 0,Y 113.965,Z 668.094,A -85,B 0,C 180,E1 -29889.363,E2 -29889.363} C_VEL
LIN {X 0,Y 102.196,Z 677.642,A -85,B 0,C 180,E1 -29891.488,E2 -29891.488} C_VEL
LIN {X 0,Y 92.3,Z 684.56,A -85,B 0,C 180,E1 -29893.876,E2 -29893.876} C_VEL
LIN {X 0,Y 80.953,Z 691.285,A -85,B 0,C 180,E1 -29897.262,E2 -29897.262} C_VEL
LIN {X 0,Y 68.45,Z 697.515,A -85,B 0,C 180,E1 -29902.474,E2 -29902.474} C_VEL
LIN {X 0,Y 56.749,Z 702.319,A -85,B 0,C 180,E1 -29909.9,E2 -29909.9} C_VEL
LIN {X 0,Y 46.42,Z 705.828,A -85,B 0,C 180,E1 -29920.801,E2 -29920.801} C_VEL
LIN {X 0,Y 38.456,Z 708.133,A -85,B 0,C 180,E1 -29936.754,E2 -29936.754} C_VEL
LIN {X 0,Y 34.385,Z 709.286,A -85,B 0,C 180,E1 -29958.208,E2 -29958.208} C_VEL
LIN {X 0,Y 34.091,Z 709.434,A -85,B 0,C 180,E1 -29970.002,E2 -29970.002} C_VEL
LIN {X 0,Y 35.847,Z 708.833,A -85,B 0,C 180,E1 -29993.088,E2 -29993.088} C_VEL
LIN {X 0,Y 42.015,Z 707.083,A -85,B 0,C 180,E1 -30011.999,E2 -30011.999} C_VEL
LIN {X 0,Y 51.322,Z 704.152,A -85,B 0,C 180,E1 -30025.251,E2 -30025.251} C_VEL
LIN {X 0,Y 51.042,Z 704.044,A -85,B 0,C 180,E1 -30026.582,E2 -30026.582} C_VEL
LIN {X 0,Y 55.662,Z 701.62,A -85,B 0,C 180,E1 -30082.259,E2 -30082.259} C_VEL
LIN {X 0,Y 58.399,Z 701.732,A -85,B 0,C 180,E1 -30088.777,E2 -30088.777} C_VEL
LIN {X 0,Y 46.449,Z 705.884,A -85,B 0,C 180,E1 -30100.839,E2 -30100.839} C_VEL
LIN {X 0,Y 38.463,Z 708.224,A -85,B 0,C 180,E1 -30116.757,E2 -30116.757} C_VEL
LIN {X 0,Y 37.488,Z 708.463,A -85,B 0,C 180,E1 -30119.894,E2 -30119.894} C_VEL
LIN {X 0,Y 35.77,Z 708.903,A -85,B 0,C 180,E1 -30125.422,E2 -30125.422} C_VEL
LIN {X 0,Y 32.908,Z 709.298,A -85,B 0,C 180,E1 -30134.098,E2 -30134.098} C_VEL
LIN {X 0,Y 27.95,Z 709.463,A -85,B 0,C 180,E1 -30159.158,E2 -30159.158} C_VEL
LIN {X 0,Y 28.21,Z 709.221,A -85,B 0,C 180,E1 -30171.481,E2 -30171.481} C_VEL
LIN {X 0,Y 28.775,Z 709.074,A -85,B 0,C 180,E1 -30175.359,E2 -30175.359} C_VEL
LIN {X 0,Y 37.012,Z 707.239,A -85,B 0,C 180,E1 -30199.422,E2 -30199.422} C_VEL
LIN {X 0,Y 47.615,Z 704.336,A -85,B 0,C 180,E1 -30212.323,E2 -30212.323} C_VEL
LIN {X 0,Y 59.691,Z 700.189,A -85,B 0,C 180,E1 -30220.374,E2 -30220.374} C_VEL
LIN {X 0,Y 72.526,Z 694.686,A -85,B 0,C 180,E1 -30225.701,E2 -30225.701} C_VEL
LIN {X 0,Y 85.82,Z 687.678,A -85,B 0,C 180,E1 -30229.326,E2 -30229.326} C_VEL
LIN {X 0,Y 96.723,Z 680.791,A -85,B 0,C 180,E1 -30231.769,E2 -30231.769} C_VEL
LIN {X 0,Y 107.858,Z 672.505,A -85,B 0,C 180,E1 -30233.556,E2 -30233.556} C_VEL
LIN {X 0,Y 118.187,Z 663.497,A -85,B 0,C 180,E1 -30234.895,E2 -30234.895} C_VEL
LIN {X 0,Y 128.572,Z 652.87,A -85,B 0,C 180,E1 -30236.007,E2 -30236.007} C_VEL
LIN {X 0,Y 138.416,Z 640.885,A -85,B 0,C 180,E1 -30236.949,E2 -30236.949} C_VEL
LIN {X 0,Y 146.829,Z 628.614,A -85,B 0,C 180,E1 -30237.68,E2 -30237.68} C_VEL
LIN {X 0,Y 154.686,Z 614.666,A -85,B 0,C 180,E1 -30238.267,E2 -30238.267} C_VEL
LIN {X 0,Y 161.247,Z 600.049,A -85,B 0,C 180,E1 -30238.682,E2 -30238.682} C_VEL
LIN {X 0,Y 166.31,Z 585.324,A -85,B 0,C 180,E1 -30238.98,E2 -30238.98} C_VEL
LIN {X 0,Y 170.089,Z 569.931,A -85,B 0,C 180,E1 -30239.203,E2 -30239.203} C_VEL
LIN {X 0,Y 172.738,Z 552.463,A -85,B 0,C 180,E1 -30239.456,E2 -30239.456} C_VEL
LIN {X 0,Y 173.248,Z 548.282,A -85,B 0,C 180,E1 -30239.559,E2 -30239.559} C_VEL
LIN {X 0,Y 173.277,Z 548.011,A -85,B 0,C 180,E1 -30240.581,E2 -30240.581} C_VEL
LIN {X 0,Y 170.526,Z 567.711,A -85,B 0,C 180,E1 -30240.827,E2 -30240.827} C_VEL
LIN {X 0,Y 167.286,Z 581.978,A -85,B 0,C 180,E1 -30241.043,E2 -30241.043} C_VEL
LIN {X 0,Y 162.432,Z 597.026,A -85,B 0,C 180,E1 -30241.33,E2 -30241.33} C_VEL
LIN {X 0,Y 156.441,Z 611.139,A -85,B 0,C 180,E1 -30241.7,E2 -30241.7} C_VEL
LIN {X 0,Y 149.451,Z 624.299,A -85,B 0,C 180,E1 -30242.162,E2 -30242.162} C_VEL
LIN {X 0,Y 140.739,Z 637.731,A -85,B 0,C 180,E1 -30242.898,E2 -30242.898} C_VEL
LIN {X 0,Y 131.183,Z 649.904,A -85,B 0,C 180,E1 -30243.79,E2 -30243.79} C_VEL
LIN {X 0,Y 121.646,Z 660.112,A -85,B 0,C 180,E1 -30244.728,E2 -30244.728} C_VEL
LIN {X 0,Y 111.307,Z 669.585,A -85,B 0,C 180,E1 -30246.032,E2 -30246.032} C_VEL
LIN {X 0,Y 99.309,Z 678.88,A -85,B 0,C 180,E1 -30247.795,E2 -30247.795} C_VEL
LIN {X 0,Y 89.174,Z 685.603,A -85,B 0,C 180,E1 -30249.887,E2 -30249.887} C_VEL
LIN {X 0,Y 75.816,Z 693.004,A -85,B 0,C 180,E1 -30253.266,E2 -30253.266} C_VEL
LIN {X 0,Y 62.853,Z 698.87,A -85,B 0,C 180,E1 -30258.116,E2 -30258.116} C_VEL
LIN {X 0,Y 53.538,Z 702.334,A -85,B 0,C 180,E1 -30263.237,E2 -30263.237} C_VEL
LIN {X 0,Y 42.102,Z 705.843,A -85,B 0,C 180,E1 -30273.424,E2 -30273.424} C_VEL
LIN {X 0,Y 32.704,Z 708.147,A -85,B 0,C 180,E1 -30289.859,E2 -30289.859} C_VEL
LIN {X 0,Y 27.463,Z 709.299,A -85,B 0,C 180,E1 -30315.175,E2 -30315.175} C_VEL
LIN {X 0,Y 26.998,Z 709.447,A -85,B 0,C 180,E1 -30330.002,E2 -30330.002} C_VEL
LIN {X 0,Y 29.42,Z 708.847,A -85,B 0,C 180,E1 -30358.542,E2 -30358.542} C_VEL
LIN {X 0,Y 37.016,Z 707.097,A -85,B 0,C 180,E1 -30379.419,E2 -30379.419} C_VEL
LIN {X 0,Y 42.097,Z 705.782,A -85,B 0,C 180,E1 -30386.591,E2 -30386.591} C_VEL
LIN {X 0,Y 42.428,Z 705.442,A -85,B 0,C 180,E1 -30390.204,E2 -30390.204} C_VEL
LIN {X 0,Y 49.347,Z 703.629,A -85,B 0,C 180,E1 -30445.295,E2 -30445.295} C_VEL
LIN {X 0,Y 47.681,Z 704.25,A -85,B 0,C 180,E1 -30447.823,E2 -30447.823} C_VEL
LIN {X 0,Y 37.029,Z 707.188,A -85,B 0,C 180,E1 -30460.605,E2 -30460.605} C_VEL
LIN {X 0,Y 29.421,Z 708.945,A -85,B 0,C 180,E1 -30481.46,E2 -30481.46} C_VEL
LIN {X 0,Y 26.99,Z 709.552,A -85,B 0,C 180,E1 -30509.998,E2 -30509.998} C_VEL
LIN {X 0,Y 28.775,Z 709.074,A -85,B 0,C 180,E1 -30535.359,E2 -30535.359} C_VEL
LIN {X 0,Y 30.637,Z 708.613,A -85,B 0,C 180,E1 -30546.126,E2 -30546.126} C_VEL
LIN {X 0,Y 34.078,Z 707.402,A -85,B 0,C 180,E1 -30562.513,E2 -30562.513} C_VEL
LIN {X 0,Y 38.248,Z 706.135,A -85,B 0,C 180,E1 -30573.125,E2 -30573.125} C_VEL
LIN {X 0,Y 42.524,Z 704.962,A -85,B 0,C 180,E1 -30578.736,E2 -30578.736} C_VEL
LIN {X 0,Y 44.171,Z 704.467,A -85,B 0,C 180,E1 -30580.074,E2 -30580.074} C_VEL
LIN {X 0,Y 54.386,Z 701.351,A -85,B 0,C 180,E1 -30585.735,E2 -30585.735} C_VEL
LIN {X 0,Y 67.713,Z 696.185,A -85,B 0,C 180,E1 -30590.401,E2 -30590.401} C_VEL
LIN {X 0,Y 81.349,Z 689.568,A -85,B 0,C 180,E1 -30593.473,E2 -30593.473} C_VEL
LIN {X 0,Y 93.866,Z 682.117,A -85,B 0,C 180,E1 -30595.706,E2 -30595.706} C_VEL
LIN {X 0,Y 105.548,Z 673.827,A -85,B 0,C 180,E1 -30597.17,E2 -30597.17} C_VEL
LIN {X 0,Y 117.767,Z 663.475,A -85,B 0,C 180,E1 -30598.355,E2 -30598.355} C_VEL
LIN {X 0,Y 128.273,Z 652.846,A -85,B 0,C 180,E1 -30599.184,E2 -30599.184} C_VEL
LIN {X 0,Y 137.596,Z 641.682,A -85,B 0,C 180,E1 -30599.859,E2 -30599.859} C_VEL
LIN {X 0,Y 139.525,Z 639.136,A -85,B 0,C 180,E1 -30600,E2 -30600} C_VEL
LIN {X 0,Y 132.659,Z 647.824,A -85,B 0,C 180,E1 -30600.567,E2 -30600.567} C_VEL
LIN {X 0,Y 123.017,Z 658.372,A -85,B 0,C 180,E1 -30601.227,E2 -30601.227} C_VEL
LIN {X 0,Y 112.528,Z 668.135,A -85,B 0,C 180,E1 -30602.176,E2 -30602.176} C_VEL
LIN {X 0,Y 100.332,Z 677.679,A -85,B 0,C 180,E1 -30603.471,E2 -30603.471} C_VEL
LIN {X 0,Y 89.939,Z 684.596,A -85,B 0,C 180,E1 -30604.932,E2 -30604.932} C_VEL
LIN {X 0,Y 81.355,Z 689.524,A -85,B 0,C 180,E1 -30606.57,E2 -30606.57} C_VEL
LIN {X 0,Y 67.723,Z 696.134,A -85,B 0,C 180,E1 -30609.647,E2 -30609.647} C_VEL
LIN {X 0,Y 54.394,Z 701.294,A -85,B 0,C 180,E1 -30614.298,E2 -30614.298} C_VEL
LIN {X 0,Y 44.765,Z 704.259,A -85,B 0,C 180,E1 -30619.615,E2 -30619.615} C_VEL
LIN {X 0,Y 32.822,Z 707.156,A -85,B 0,C 180,E1 -30631.076,E2 -30631.076} C_VEL
LIN {X 0,Y 23.408,Z 708.88,A -85,B 0,C 180,E1 -30653.099,E2 -30653.099} C_VEL
LIN {X 0,Y 19.894,Z 709.461,A -85,B 0,C 180,E1 -30690.003,E2 -30690.003} C_VEL
LIN {X 0,Y 23.409,Z 708.86,A -85,B 0,C 180,E1 -30726.904,E2 -30726.904} C_VEL
LIN {X 0,Y 32.823,Z 707.11,A -85,B 0,C 180,E1 -30748.927,E2 -30748.927} C_VEL
LIN {X 0,Y 34.442,Z 706.688,A -85,B 0,C 180,E1 -30753.258,E2 -30753.258} C_VEL
LIN {X 0,Y 39.022,Z 705.594,A -85,B 0,C 180,E1 -30801.114,E2 -30801.114} C_VEL
LIN {X 0,Y 38.646,Z 705.857,A -85,B 0,C 180,E1 -30804.592,E2 -30804.592} C_VEL
LIN {X 0,Y 27.627,Z 708.197,A -85,B 0,C 180,E1 -30820.253,E2 -30820.253} C_VEL
LIN {X 0,Y 20.614,Z 709.382,A -85,B 0,C 180,E1 -30850.064,E2 -30850.064} C_VEL
LIN {X 0,Y 19.884,Z 709.538,A -85,B 0,C 180,E1 -30869.997,E2 -30869.997} C_VEL
LIN {X 0,Y 23.407,Z 708.953,A -85,B 0,C 180,E1 -30906.902,E2 -30906.902} C_VEL
LIN {X 0,Y 32.819,Z 707.224,A -85,B 0,C 180,E1 -30928.93,E2 -30928.93} C_VEL
LIN {X 0,Y 44.171,Z 704.467,A -85,B 0,C 180,E1 -30940.074,E2 -30940.074} C_VEL
LIN {X 0,Y 48.987,Z 703.082,A -85,B 0,C 180,E1 -30943.941,E2 -30943.941} C_VEL
LIN {X 0,Y 56.457,Z 700.431,A -85,B 0,C 180,E1 -30950.452,E2 -30950.452} C_VEL
LIN {X 0,Y 62.673,Z 697.937,A -85,B 0,C 180,E1 -30954.588,E2 -30954.588} C_VEL
LIN {X 0,Y 67.723,Z 695.832,A -85,B 0,C 180,E1 -30956.555,E2 -30956.555} C_VEL
LIN {X 0,Y 69.484,Z 695.039,A -85,B 0,C 180,E1 -30956.938,E2 -30956.938} C_VEL
LIN {X 0,Y 80.848,Z 689.551,A -85,B 0,C 180,E1 -30958.513,E2 -30958.513} C_VEL
LIN {X 0,Y 92.748,Z 682.637,A -85,B 0,C 180,E1 -30960,E2 -30960} C_VEL
LIN {X 0,Y 80.85,Z 689.541,A -85,B 0,C 180,E1 -30961.52,E2 -30961.52} C_VEL
LIN {X 0,Y 66.897,Z 696.15,A -85,B 0,C 180,E1 -30963.592,E2 -30963.592} C_VEL
LIN {X 0,Y 53.082,Z 701.309,A -85,B 0,C 180,E1 -30966.792,E2 -30966.792} C_VEL
LIN {X 0,Y 42.897,Z 704.273,A -85,B 0,C 180,E1 -30970.585,E2 -30970.585} C_VEL
LIN {X 0,Y 29.773,Z 707.17,A -85,B 0,C 180,E1 -30979.235,E2 -30979.235} C_VEL
LIN {X 0,Y 18.202,Z 708.894,A -85,B 0,C 180,E1 -30999.449,E2 -30999.449} C_VEL
LIN {X 0,Y 12.782,Z 709.475,A -85,B 0,C 180,E1 -31050.004,E2 -31050.004} C_VEL
LIN {X 0,Y 18.203,Z 708.874,A -85,B 0,C 180,E1 -31100.554,E2 -31100.554} C_VEL
LIN {X 0,Y 25.403,Z 707.902,A -85,B 0,C 180,E1 -31115.754,E2 -31115.754} C_VEL
LIN {X 0,Y 26.199,Z 707.585,A -85,B 0,C 180,E1 -31124.441,E2 -31124.441} C_VEL
LIN {X 0,Y 29.156,Z 707.157,A -85,B 0,C 180,E1 -31155.375,E2 -31155.375} C_VEL
LIN {X 0,Y 29.783,Z 707.161,A -85,B 0,C 180,E1 -31159.278,E2 -31159.278} C_VEL
LIN {X 0,Y 18.205,Z 708.918,A -85,B 0,C 180,E1 -31179.454,E2 -31179.454} C_VEL
LIN {X 0,Y 12.772,Z 709.524,A -85,B 0,C 180,E1 -31229.996,E2 -31229.996} C_VEL
LIN {X 0,Y 18.201,Z 708.939,A -85,B 0,C 180,E1 -31280.554,E2 -31280.554} C_VEL
LIN {X 0,Y 29.771,Z 707.21,A -85,B 0,C 180,E1 -31300.776,E2 -31300.776} C_VEL
LIN {X 0,Y 42.878,Z 704.306,A -85,B 0,C 180,E1 -31309.549,E2 -31309.549} C_VEL
LIN {X 0,Y 56.516,Z 700.158,A -85,B 0,C 180,E1 -31314.167,E2 -31314.167} C_VEL
LIN {X 0,Y 69.484,Z 695.039,A -85,B 0,C 180,E1 -31316.938,E2 -31316.938} C_VEL
LIN {X 0,Y 68.197,Z 695.609,A -85,B 0,C 180,E1 -31317.711,E2 -31317.711} C_VEL
LIN {X 0,Y 64.135,Z 697.28,A -85,B 0,C 180,E1 -31318.41,E2 -31318.41} C_VEL
LIN {X 0,Y 54.627,Z 700.71,A -85,B 0,C 180,E1 -31318.943,E2 -31318.943} C_VEL
LIN {X 0,Y 48.343,Z 702.639,A -85,B 0,C 180,E1 -31319.045,E2 -31319.045} C_VEL
LIN {X 0,Y 42.028,Z 704.33,A -85,B 0,C 180,E1 -31318.717,E2 -31318.717} C_VEL
LIN {X 0,Y 35.722,Z 705.769,A -85,B 0,C 180,E1 -31317.463,E2 -31317.463} C_VEL
LIN {X 0,Y 21.377,Z 708.204,A -85,B 0,C 180,E1 -31310.496,E2 -31310.496} C_VEL
LIN {X 0,Y 8.708,Z 709.361,A -85,B 0,C 180,E1 -31283.8,E2 -31283.8} C_VEL
LIN {X 0,Y 5.673,Z 709.51,A -85,B 0,C 180,E1 -31229.991,E2 -31229.991} C_VEL
LIN {X 0,Y 14.735,Z 708.904,A -85,B 0,C 180,E1 -31157.448,E2 -31157.448} C_VEL
LIN {X 0,Y 17.238,Z 708.661,A -85,B 0,C 180,E1 -31153.748,E2 -31153.748} C_VEL
LIN {X 0,Y 19.949,Z 708.307,A -85,B 0,C 180,E1 -31145.895,E2 -31145.895} C_VEL
LIN {X 0,Y 19.14,Z 708.391,A -85,B 0,C 180,E1 -31133.867,E2 -31133.867} C_VEL
LIN {X 0,Y 18.32,Z 708.517,A -85,B 0,C 180,E1 -31127.522,E2 -31127.522} C_VEL
LIN {X 0,Y 8.726,Z 709.334,A -85,B 0,C 180,E1 -31103.657,E2 -31103.657} C_VEL
LIN {X 0,Y 5.683,Z 709.489,A -85,B 0,C 180,E1 -31050.009,E2 -31050.009} C_VEL
LIN {X 0,Y 14.732,Z 708.908,A -85,B 0,C 180,E1 -30977.434,E2 -30977.434} C_VEL
LIN {X 0,Y 28.238,Z 707.185,A -85,B 0,C 180,E1 -30965.439,E2 -30965.439} C_VEL
LIN {X 0,Y 42.173,Z 704.288,A -85,B 0,C 180,E1 -30960.965,E2 -30960.965} C_VEL
LIN {X 0,Y 45.935,Z 703.339,A -85,B 0,C 180,E1 -30959.999,E2 -30959.999} C_VEL
LIN {X 0,Y 35.722,Z 705.769,A -85,B 0,C 180,E1 -30957.463,E2 -30957.463} C_VEL
LIN {X 0,Y 35.722,Z 705.769,A -85,B 0,C 180,E1 -30957.463,E2 -30957.463}

QRS_NEXT_CUT()

QRS_NEXT()
QRS_HOME()

END
